KUKA KRL program: FINA11.src

&ACCESS RVP
&REL 143
DEF FINA11()
   DECL E6axis PX1 ;shengming px1 bianliang

   GLOBAL INTERRUPT DECL 3 WHEN $STOPMESS==TRUE DO IR_STOPM ( )
   INTERRUPT ON 3
   BAS (#INITMOV,0)
   BAS (#VEL_PTP,20)
   BAS (#ACC_PTP,20)
   $APO.CDIS = 100.0
   $VEL.CP = 0.5
   $ADVANCE=5
   $TOOL={X 0, Y 0, Z 319.5, A 0, B 0, C 0}
   $BASE={X 1708, Y 89, Z 1050, A 180, B 0, C 180}
   PTP {A1 -30.000, A2 -120.000, A3 120.000, A4 0.000, A5 0.000, A6 0.000, E1 0, E2 0, E3 0, E4 0, E5 0, E6 0}
   $async_EX_AX_DECOUPLE='b0001' ;dianji qu ouhe
   $AXIS_ACT.E1=0 ;bianmqi qingling
   WAIT SEC 1 ; yanshi 1s
   $async_EX_AX_DECOUPLE='b0000' ;dianji ouhe
   HALT
   $advance=5
   $VEL.CP=0.167
   $APO.CDIS = 0
   CONTINUE ;dongzuo lianguan
   ;IF SELT_MODE==1 THEN
   PTP {A1 5, A2 -84.46, A3 114.11, A4 59.82, A5 -48.27, A6 67.3, E1 0, E2 0, E3 0, E4 0, E5 0, E6 0} ;fenxian weizhi
   PTP {A1 5, A2 -84.46, A3 114.11, A4 59.82, A5 -48.27, A6 67.3, E1 0, E2 0, E3 0, E4 0, E5 0, E6 0} ;fenxian weizhi
   HALT ;zanting
   $APO.CDIS = 100 ;yuanhuaguodu
   PX1=$AXIS_ACT ;jiang dang qian jiaodu fuzhi gei px1
   NUM_TURN=1  ;zhuan jiao du ji shu bian liang
   CONTINUE
   $VEL.CP=0.167
   FOR NUM_TURN=1 TO 30  ;jiang NUM_TURN bianliang xunhuan 10ci
      PX1.E1=PX1.E1+120.0
      PTP PX1 C_DIS ;
   ENDFOR
   ;zan ting
   HALT
   ;PTP {A1 2.39, A2 -82.14, A3 104.12, A4 65.48, A5 -43.86, A6 58.47, E1 -84.06, E2 0, E3 0, E4 0, E5 0, E6 0}

   ;ELSE
   ;PTP {A1 7.433, A2 -36.447, A3 70.255, A4 38.782, A5 -95.202, A6 0.000, E1 -55.75, E2 0, E3 0, E4 0, E5 0, E6 0}
   ;SPTP {A1 7.433, A2 -36.447, A3 70.255, A4 38.782, A5 -95.202, A6 0.000, E1 -55.75, E2 0, E3 0, E4 0, E5 0, E6 0} C_DIS
   ;Start
   $VEL.CP=0.133
   SPTP {A1 7.880, A2 -36.991, A3 70.406, A4 40.976, A5 -94.486, A6 0.000, E1 -55.64, E2 0, E3 0, E4 0, E5 0, E6 0} C_DIS
   SPTP {A1 8.283, A2 -37.781, A3 70.980, A4 43.029, A5 -93.598, A6 0.000, E1 -55.77, E2 0, E3 0, E4 0, E5 0, E6 0} C_DIS
   SPTP {A1 8.645, A2 -38.809, A3 71.949, A4 44.960, A5 -92.527, A6 0.000, E1 -56.19, E2 0, E3 0, E4 0, E5 0, E6 0} C_DIS
   SPTP {A1 9.000, A2 -39.796, A3 72.797, A4 46.914, A5 -91.440, A6 0.000, E1 -56.68, E2 0, E3 0, E4 0, E5 0, E6 0} C_DIS
   SPTP {A1 9.348, A2 -40.751, A3 73.545, A4 48.891, A5 -90.338, A6 0.000, E1 -57.25, E2 0, E3 0, E4 0, E5 0, E6 0} C_DIS
   SPTP {A1 9.684, A2 -41.681, A3 74.210, A4 50.878, A5 -89.222, A6 0.000, E1 -57.87, E2 0, E3 0, E4 0, E5 0, E6 0} C_DIS
   SPTP {A1 10.009, A2 -42.594, A3 74.803, A4 52.874, A5 -88.090, A6 0.000, E1 -58.54, E2 0, E3 0, E4 0, E5 0, E6 0} C_DIS
   SPTP {A1 10.320, A2 -43.493, A3 75.334, A4 54.874, A5 -86.941, A6 0.000, E1 -59.25, E2 0, E3 0, E4 0, E5 0, E6 0} C_DIS
   SPTP {A1 10.615, A2 -44.382, A3 75.814, A4 56.876, A5 -85.776, A6 0.000, E1 -60, E2 0, E3 0, E4 0, E5 0, E6 0} C_DIS
   SPTP {A1 10.870, A2 -45.375, A3 76.460, A4 58.776, A5 -84.526, A6 0.000, E1 -60.98, E2 0, E3 0, E4 0, E5 0, E6 0} C_DIS
   SPTP {A1 11.099, A2 -46.403, A3 77.133, A4 60.647, A5 -83.228, A6 0.000, E1 -62.08, E2 0, E3 0, E4 0, E5 0, E6 0} C_DIS
   SPTP {A1 11.315, A2 -47.400, A3 77.716, A4 62.556, A5 -81.937, A6 0.000, E1 -63.25, E2 0, E3 0, E4 0, E5 0, E6 0} C_DIS
   SPTP {A1 11.512, A2 -48.390, A3 78.250, A4 64.480, A5 -80.631, A6 0.000, E1 -64.49, E2 0, E3 0, E4 0, E5 0, E6 0} C_DIS
   SPTP {A1 11.690, A2 -49.362, A3 78.719, A4 66.433, A5 -79.325, A6 0.000, E1 -65.79, E2 0, E3 0, E4 0, E5 0, E6 0} C_DIS
   SPTP {A1 11.848, A2 -50.324, A3 79.141, A4 68.407, A5 -78.011, A6 0.000, E1 -67.16, E2 0, E3 0, E4 0, E5 0, E6 0} C_DIS
   SPTP {A1 11.984, A2 -51.273, A3 79.509, A4 70.411, A5 -76.698, A6 0.000, E1 -68.6, E2 0, E3 0, E4 0, E5 0, E6 0} C_DIS
   SPTP {A1 12.098, A2 -52.202, A3 79.819, A4 72.452, A5 -75.397, A6 0.000, E1 -70.12, E2 0, E3 0, E4 0, E5 0, E6 0} C_DIS
   SPTP {A1 12.187, A2 -53.119, A3 80.083, A4 74.527, A5 -74.100, A6 0.000, E1 -71.71, E2 0, E3 0, E4 0, E5 0, E6 0} C_DIS
   SPTP {A1 12.253, A2 -54.007, A3 80.279, A4 76.654, A5 -72.833, A6 0.000, E1 -73.4, E2 0, E3 0, E4 0, E5 0, E6 0} C_DIS
   SPTP {A1 12.292, A2 -54.883, A3 80.432, A4 78.822, A5 -71.578, A6 0.000, E1 -75.17, E2 0, E3 0, E4 0, E5 0, E6 0} C_DIS
   SPTP {A1 12.307, A2 -55.719, A3 80.506, A4 81.058, A5 -70.379, A6 0.000, E1 -77.05, E2 0, E3 0, E4 0, E5 0, E6 0} C_DIS
   SPTP {A1 12.293, A2 -56.537, A3 80.534, A4 83.344, A5 -69.206, A6 0.000, E1 -79.02, E2 0, E3 0, E4 0, E5 0, E6 0} C_DIS
   SPTP {A1 12.254, A2 -57.299, A3 80.488, A4 85.654, A5 -68.116, A6 0.000, E1 -81, E2 0, E3 0, E4 0, E5 0, E6 0} C_DIS
   SPTP {A1 12.184, A2 -57.979, A3 80.434, A4 87.746, A5 -67.107, A6 0.000, E1 -82.51, E2 0, E3 0, E4 0, E5 0, E6 0} C_DIS
   HALT
   SPTP {A1 12.090, A2 -58.636, A3 80.350, A4 89.865, A5 -66.133, A6 0.000, E1 -84.06, E2 0, E3 0, E4 0, E5 0, E6 0} C_DIS
   SPTP {A1 11.972, A2 -59.275, A3 80.235, A4 92.031, A5 -65.193, A6 0.000, E1 -85.68, E2 0, E3 0, E4 0, E5 0, E6 0} C_DIS
   SPTP {A1 11.830, A2 -59.891, A3 80.084, A4 94.249, A5 -64.297, A6 0.000, E1 -87.37, E2 0, E3 0, E4 0, E5 0, E6 0} C_DIS
   SPTP {A1 11.665, A2 -60.478, A3 79.890, A4 96.525, A5 -63.457, A6 0.000, E1 -89.15, E2 0, E3 0, E4 0, E5 0, E6 0} C_DIS
   SPTP {A1 11.477, A2 -61.034, A3 79.651, A4 98.858, A5 -62.682, A6 0.000, E1 -91.01, E2 0, E3 0, E4 0, E5 0, E6 0} C_DIS
   SPTP {A1 11.269, A2 -61.552, A3 79.358, A4 101.252, A5 -61.990, A6 0.000, E1 -92.95, E2 0, E3 0, E4 0, E5 0, E6 0} C_DIS
   SPTP {A1 11.041, A2 -62.032, A3 79.039, A4 103.636, A5 -61.365, A6 0.000, E1 -94.82, E2 0, E3 0, E4 0, E5 0, E6 0} C_DIS
   SPTP {A1 10.795, A2 -62.519, A3 78.970, A4 105.496, A5 -60.574, A6 0.000, E1 -95.67, E2 0, E3 0, E4 0, E5 0, E6 0} C_DIS
   SPTP {A1 10.532, A2 -62.995, A3 78.892, A4 107.395, A5 -59.807, A6 0.000, E1 -96.57, E2 0, E3 0, E4 0, E5 0, E6 0} C_DIS
   SPTP {A1 10.254, A2 -63.455, A3 78.799, A4 109.336, A5 -59.075, A6 0.000, E1 -97.51, E2 0, E3 0, E4 0, E5 0, E6 0} C_DIS
   SPTP {A1 9.963, A2 -63.890, A3 78.682, A4 111.320, A5 -58.395, A6 0.000, E1 -98.5, E2 0, E3 0, E4 0, E5 0, E6 0} C_DIS
   SPTP {A1 9.661, A2 -64.298, A3 78.535, A4 113.347, A5 -57.779, A6 0.000, E1 -99.53, E2 0, E3 0, E4 0, E5 0, E6 0} C_DIS
   SPTP {A1 9.351, A2 -64.674, A3 78.354, A4 115.414, A5 -57.239, A6 0.000, E1 -100.59, E2 0, E3 0, E4 0, E5 0, E6 0} C_DIS
   SPTP {A1 9.036, A2 -65.116, A3 78.480, A4 117.001, A5 -56.418, A6 0.000, E1 -100.81, E2 0, E3 0, E4 0, E5 0, E6 0} C_DIS
   SPTP {A1 8.718, A2 -65.623, A3 78.879, A4 118.187, A5 -55.327, A6 0.000, E1 -100.36, E2 0, E3 0, E4 0, E5 0, E6 0} C_DIS
   SPTP {A1 8.399, A2 -66.115, A3 79.274, A4 119.383, A5 -54.253, A6 0.000, E1 -99.91, E2 0, E3 0, E4 0, E5 0, E6 0} C_DIS
   SPTP {A1 8.080, A2 -66.590, A3 79.662, A4 120.587, A5 -53.203, A6 0.000, E1 -99.46, E2 0, E3 0, E4 0, E5 0, E6 0} C_DIS
   SPTP {A1 7.762, A2 -67.048, A3 80.044, A4 121.798, A5 -52.179, A6 0.000, E1 -99.01, E2 0, E3 0, E4 0, E5 0, E6 0} C_DIS
   SPTP {A1 7.452, A2 -67.536, A3 80.590, A4 122.724, A5 -50.992, A6 0.000, E1 -98.13, E2 0, E3 0, E4 0, E5 0, E6 0} C_DIS
   SPTP {A1 7.154, A2 -68.181, A3 81.750, A4 122.572, A5 -49.106, A6 0.000, E1 -95.74, E2 0, E3 0, E4 0, E5 0, E6 0} C_DIS
   SPTP {A1 6.864, A2 -68.792, A3 82.894, A4 122.305, A5 -47.234, A6 0.000, E1 -93.25, E2 0, E3 0, E4 0, E5 0, E6 0} C_DIS
   SPTP {A1 6.585, A2 -69.369, A3 84.019, A4 121.908, A5 -45.386, A6 0.000, E1 -90.65, E2 0, E3 0, E4 0, E5 0, E6 0} C_DIS
   SPTP {A1 6.318, A2 -69.912, A3 85.124, A4 121.367, A5 -43.568, A6 0.000, E1 -87.91, E2 0, E3 0, E4 0, E5 0, E6 0} C_DIS
   SPTP {A1 6.068, A2 -70.459, A3 86.414, A4 120.139, A5 -41.551, A6 0.000, E1 -84.38, E2 0, E3 0, E4 0, E5 0, E6 0} C_DIS
   SPTP {A1 5.835, A2 -71.046, A3 88.208, A4 117.103, A5 -39.004, A6 0.000, E1 -78.78, E2 0, E3 0, E4 0, E5 0, E6 0} C_DIS
   SPTP {A1 5.615, A2 -71.534, A3 89.916, A4 113.493, A5 -36.647, A6 0.000, E1 -72.65, E2 0, E3 0, E4 0, E5 0, E6 0} C_DIS
   SPTP {A1 5.408, A2 -71.925, A3 91.535, A4 109.257, A5 -34.526, A6 0.000, E1 -65.93, E2 0, E3 0, E4 0, E5 0, E6 0} C_DIS
   SPTP {A1 5.213, A2 -72.216, A3 93.061, A4 104.367, A5 -32.693, A6 0.000, E1 -58.59, E2 0, E3 0, E4 0, E5 0, E6 0} C_DIS
   SPTP {A1 5.032, A2 -72.407, A3 94.490, A4 98.837, A5 -31.209, A6 0.000, E1 -50.64, E2 0, E3 0, E4 0, E5 0, E6 0} C_DIS
   SPTP {A1 4.862, A2 -72.471, A3 95.949, A4 91.902, A5 -30.163, A6 0.000, E1 -41.35, E2 0, E3 0, E4 0, E5 0, E6 0} C_DIS
   SPTP {A1 4.701, A2 -72.389, A3 97.348, A4 84.053, A5 -29.733, A6 0.000, E1 -31.19, E2 0, E3 0, E4 0, E5 0, E6 0} C_DIS
   SPTP {A1 4.547, A2 -72.174, A3 98.598, A4 76.137, A5 -29.944, A6 0.000, E1 -20.99, E2 0, E3 0, E4 0, E5 0, E6 0} C_DIS
   SPTP {A1 4.399, A2 -71.829, A3 99.695, A4 68.521, A5 -30.775, A6 0.000, E1 -11.11, E2 0, E3 0, E4 0, E5 0, E6 0} C_DIS
   SPTP {A1 4.261, A2 -71.353, A3 100.632, A4 61.519, A5 -32.180, A6 0.000, E1 -1.84, E2 0, E3 0, E4 0, E5 0, E6 0} C_DIS
   SPTP {A1 4.136, A2 -70.751, A3 101.404, A4 55.307, A5 -34.070, A6 0.000, E1 6.63, E2 0, E3 0, E4 0, E5 0, E6 0} C_DIS
   SPTP {A1 4.022, A2 -70.030, A3 102.012, A4 49.932, A5 -36.348, A6 0.000, E1 14.27, E2 0, E3 0, E4 0, E5 0, E6 0} C_DIS
   SPTP {A1 3.922, A2 -69.194, A3 102.450, A4 45.377, A5 -38.927, A6 0.000, E1 21.11, E2 0, E3 0, E4 0, E5 0, E6 0} C_DIS
   SPTP {A1 3.840, A2 -68.251, A3 102.716, A4 41.575, A5 -41.730, A6 0.000, E1 27.21, E2 0, E3 0, E4 0, E5 0, E6 0} C_DIS
   SPTP {A1 3.776, A2 -67.320, A3 102.827, A4 38.663, A5 -44.407, A6 0.000, E1 32.35, E2 0, E3 0, E4 0, E5 0, E6 0} C_DIS
   SPTP {A1 3.725, A2 -66.575, A3 102.861, A4 36.670, A5 -46.536, A6 0.000, E1 36.37, E2 0, E3 0, E4 0, E5 0, E6 0} C_DIS
   SPTP {A1 3.694, A2 -65.782, A3 102.799, A4 34.989, A5 -48.712, A6 0.000, E1 40.11, E2 0, E3 0, E4 0, E5 0, E6 0} C_DIS
   SPTP {A1 3.683, A2 -64.947, A3 102.644, A4 33.590, A5 -50.918, A6 0.000, E1 43.61, E2 0, E3 0, E4 0, E5 0, E6 0} C_DIS
   SPTP {A1 3.692, A2 -64.071, A3 102.395, A4 32.447, A5 -53.136, A6 0.000, E1 46.88, E2 0, E3 0, E4 0, E5 0, E6 0} C_DIS
   SPTP {A1 3.720, A2 -63.161, A3 102.055, A4 31.529, A5 -55.351, A6 0.000, E1 49.96, E2 0, E3 0, E4 0, E5 0, E6 0} C_DIS
   SPTP {A1 3.765, A2 -62.219, A3 101.624, A4 30.813, A5 -57.551, A6 0.000, E1 52.88, E2 0, E3 0, E4 0, E5 0, E6 0} C_DIS
   SPTP {A1 3.868, A2 -61.648, A3 101.314, A4 30.672, A5 -58.896, A6 0.000, E1 55.21, E2 0, E3 0, E4 0, E5 0, E6 0} C_DIS
   SPTP {A1 3.996, A2 -61.138, A3 100.997, A4 30.721, A5 -60.077, A6 0.000, E1 57.38, E2 0, E3 0, E4 0, E5 0, E6 0} C_DIS
   SPTP {A1 4.141, A2 -60.619, A3 100.641, A4 30.875, A5 -61.247, A6 0.000, E1 59.47, E2 0, E3 0, E4 0, E5 0, E6 0} C_DIS
   SPTP {A1 4.300, A2 -60.092, A3 100.246, A4 31.122, A5 -62.400, A6 0.000, E1 61.49, E2 0, E3 0, E4 0, E5 0, E6 0} C_DIS
   SPTP {A1 4.471, A2 -59.559, A3 99.814, A4 31.448, A5 -63.534, A6 0.000, E1 63.46, E2 0, E3 0, E4 0, E5 0, E6 0} C_DIS
   SPTP {A1 4.653, A2 -59.019, A3 99.345, A4 31.854, A5 -64.648, A6 0.000, E1 65.37, E2 0, E3 0, E4 0, E5 0, E6 0} C_DIS
   SPTP {A1 4.843, A2 -58.475, A3 98.842, A4 32.326, A5 -65.738, A6 0.000, E1 67.23, E2 0, E3 0, E4 0, E5 0, E6 0} C_DIS
   SPTP {A1 5.048, A2 -57.962, A3 98.326, A4 32.894, A5 -66.735, A6 0.000, E1 69.02, E2 0, E3 0, E4 0, E5 0, E6 0} C_DIS
   SPTP {A1 5.321, A2 -57.796, A3 98.000, A4 33.874, A5 -67.052, A6 0.000, E1 70.48, E2 0, E3 0, E4 0, E5 0, E6 0} C_DIS
   SPTP {A1 5.599, A2 -57.626, A3 97.650, A4 34.901, A5 -67.358, A6 0.000, E1 71.89, E2 0, E3 0, E4 0, E5 0, E6 0} C_DIS
   SPTP {A1 5.882, A2 -57.453, A3 97.275, A4 35.972, A5 -67.654, A6 0.000, E1 73.26, E2 0, E3 0, E4 0, E5 0, E6 0} C_DIS
   SPTP {A1 6.166, A2 -57.278, A3 96.877, A4 37.078, A5 -67.938, A6 0.000, E1 74.59, E2 0, E3 0, E4 0, E5 0, E6 0} C_DIS
   SPTP {A1 6.452, A2 -57.099, A3 96.455, A4 38.215, A5 -68.213, A6 0.000, E1 75.9, E2 0, E3 0, E4 0, E5 0, E6 0} C_DIS
   SPTP {A1 6.737, A2 -56.918, A3 96.010, A4 39.378, A5 -68.477, A6 0.000, E1 77.18, E2 0, E3 0, E4 0, E5 0, E6 0} C_DIS
   SPTP {A1 7.020, A2 -56.735, A3 95.545, A4 40.563, A5 -68.731, A6 0.000, E1 78.43, E2 0, E3 0, E4 0, E5 0, E6 0} C_DIS
   SPTP {A1 7.301, A2 -56.550, A3 95.058, A4 41.765, A5 -68.973, A6 0.000, E1 79.67, E2 0, E3 0, E4 0, E5 0, E6 0} C_DIS
   SPTP {A1 7.577, A2 -56.363, A3 94.553, A4 42.980, A5 -69.205, A6 0.000, E1 80.88, E2 0, E3 0, E4 0, E5 0, E6 0} C_DIS
   SPTP {A1 7.849, A2 -56.176, A3 94.029, A4 44.204, A5 -69.426, A6 0.000, E1 82.08, E2 0, E3 0, E4 0, E5 0, E6 0} C_DIS
   SPTP {A1 8.115, A2 -55.987, A3 93.489, A4 45.437, A5 -69.637, A6 0.000, E1 83.27, E2 0, E3 0, E4 0, E5 0, E6 0} C_DIS
   SPTP {A1 8.380, A2 -55.851, A3 92.971, A4 46.723, A5 -69.748, A6 0.000, E1 84.36, E2 0, E3 0, E4 0, E5 0, E6 0} C_DIS
   SPTP {A1 8.645, A2 -55.786, A3 92.489, A4 48.086, A5 -69.733, A6 0.000, E1 85.33, E2 0, E3 0, E4 0, E5 0, E6 0} C_DIS
   SPTP {A1 8.902, A2 -55.719, A3 91.992, A4 49.451, A5 -69.712, A6 0.000, E1 86.28, E2 0, E3 0, E4 0, E5 0, E6 0} C_DIS
   SPTP {A1 9.152, A2 -55.650, A3 91.480, A4 50.817, A5 -69.688, A6 0.000, E1 87.22, E2 0, E3 0, E4 0, E5 0, E6 0} C_DIS
   SPTP {A1 9.393, A2 -55.581, A3 90.956, A4 52.180, A5 -69.658, A6 0.000, E1 88.15, E2 0, E3 0, E4 0, E5 0, E6 0} C_DIS
   SPTP {A1 9.624, A2 -55.511, A3 90.422, A4 53.538, A5 -69.624, A6 0.000, E1 89.08, E2 0, E3 0, E4 0, E5 0, E6 0} C_DIS
   SPTP {A1 9.845, A2 -55.443, A3 89.880, A4 54.890, A5 -69.583, A6 0.000, E1 90, E2 0, E3 0, E4 0, E5 0, E6 0} C_DIS
   SPTP {A1 10.057, A2 -55.377, A3 89.331, A4 56.233, A5 -69.536, A6 0.000, E1 90.92, E2 0, E3 0, E4 0, E5 0, E6 0} C_DIS
   SPTP {A1 10.258, A2 -55.314, A3 88.779, A4 57.563, A5 -69.480, A6 0.000, E1 91.84, E2 0, E3 0, E4 0, E5 0, E6 0} C_DIS
   SPTP {A1 10.448, A2 -55.255, A3 88.225, A4 58.882, A5 -69.417, A6 0.000, E1 92.76, E2 0, E3 0, E4 0, E5 0, E6 0} C_DIS
   SPTP {A1 10.623, A2 -55.202, A3 87.683, A4 60.164, A5 -69.349, A6 0.000, E1 93.68, E2 0, E3 0, E4 0, E5 0, E6 0} C_DIS
   SPTP {A1 10.779, A2 -55.156, A3 87.166, A4 61.385, A5 -69.290, A6 0.000, E1 94.58, E2 0, E3 0, E4 0, E5 0, E6 0} C_DIS
   SPTP {A1 10.910, A2 -55.118, A3 86.689, A4 62.513, A5 -69.244, A6 0.000, E1 95.46, E2 0, E3 0, E4 0, E5 0, E6 0} C_DIS
   SPTP {A1 11.018, A2 -55.088, A3 86.256, A4 63.546, A5 -69.214, A6 0.000, E1 96.32, E2 0, E3 0, E4 0, E5 0, E6 0} C_DIS
   SPTP {A1 11.118, A2 -55.067, A3 85.835, A4 64.562, A5 -69.171, A6 0.000, E1 97.19, E2 0, E3 0, E4 0, E5 0, E6 0} C_DIS
   SPTP {A1 11.209, A2 -55.057, A3 85.426, A4 65.558, A5 -69.111, A6 0.000, E1 98.08, E2 0, E3 0, E4 0, E5 0, E6 0} C_DIS
   SPTP {A1 11.292, A2 -55.060, A3 85.035, A4 66.532, A5 -69.032, A6 0.000, E1 98.98, E2 0, E3 0, E4 0, E5 0, E6 0} C_DIS
   SPTP {A1 11.366, A2 -55.075, A3 84.661, A4 67.487, A5 -68.936, A6 0.000, E1 99.9, E2 0, E3 0, E4 0, E5 0, E6 0} C_DIS
   SPTP {A1 11.432, A2 -55.102, A3 84.304, A4 68.421, A5 -68.820, A6 0.000, E1 100.83, E2 0, E3 0, E4 0, E5 0, E6 0} C_DIS
   SPTP {A1 11.490, A2 -55.143, A3 83.969, A4 69.335, A5 -68.684, A6 0.000, E1 101.78, E2 0, E3 0, E4 0, E5 0, E6 0} C_DIS
   SPTP {A1 11.539, A2 -55.199, A3 83.655, A4 70.227, A5 -68.526, A6 0.000, E1 102.74, E2 0, E3 0, E4 0, E5 0, E6 0} C_DIS
   SPTP {A1 11.581, A2 -55.269, A3 83.364, A4 71.100, A5 -68.347, A6 0.000, E1 103.72, E2 0, E3 0, E4 0, E5 0, E6 0} C_DIS
   SPTP {A1 11.614, A2 -55.358, A3 83.100, A4 71.948, A5 -68.140, A6 0.000, E1 104.71, E2 0, E3 0, E4 0, E5 0, E6 0} C_DIS
   SPTP {A1 11.638, A2 -55.462, A3 82.861, A4 72.775, A5 -67.908, A6 0.000, E1 105.72, E2 0, E3 0, E4 0, E5 0, E6 0} C_DIS
   SPTP {A1 11.655, A2 -55.583, A3 82.649, A4 73.581, A5 -67.651, A6 0.000, E1 106.75, E2 0, E3 0, E4 0, E5 0, E6 0} C_DIS
   SPTP {A1 11.664, A2 -55.722, A3 82.465, A4 74.365, A5 -67.366, A6 0.000, E1 107.8, E2 0, E3 0, E4 0, E5 0, E6 0} C_DIS
   SPTP {A1 11.664, A2 -55.877, A3 82.310, A4 75.127, A5 -67.054, A6 0.000, E1 108.86, E2 0, E3 0, E4 0, E5 0, E6 0} C_DIS
   SPTP {A1 11.657, A2 -56.050, A3 82.184, A4 75.868, A5 -66.713, A6 0.000, E1 109.94, E2 0, E3 0, E4 0, E5 0, E6 0} C_DIS
   SPTP {A1 11.642, A2 -56.241, A3 82.087, A4 76.588, A5 -66.342, A6 0.000, E1 111.03, E2 0, E3 0, E4 0, E5 0, E6 0} C_DIS
   SPTP {A1 11.614, A2 -56.480, A3 82.054, A4 77.308, A5 -65.925, A6 0.000, E1 111.95, E2 0, E3 0, E4 0, E5 0, E6 0} C_DIS
   SPTP {A1 11.575, A2 -56.756, A3 82.072, A4 78.027, A5 -65.467, A6 0.000, E1 112.75, E2 0, E3 0, E4 0, E5 0, E6 0} C_DIS
   SPTP {A1 11.529, A2 -57.044, A3 82.112, A4 78.732, A5 -64.986, A6 0.000, E1 113.55, E2 0, E3 0, E4 0, E5 0, E6 0} C_DIS
   SPTP {A1 11.475, A2 -57.347, A3 82.174, A4 79.421, A5 -64.478, A6 0.000, E1 114.36, E2 0, E3 0, E4 0, E5 0, E6 0} C_DIS
   SPTP {A1 11.413, A2 -57.663, A3 82.259, A4 80.095, A5 -63.943, A6 0.000, E1 115.18, E2 0, E3 0, E4 0, E5 0, E6 0} C_DIS
   SPTP {A1 11.344, A2 -57.991, A3 82.364, A4 80.756, A5 -63.383, A6 0.000, E1 116, E2 0, E3 0, E4 0, E5 0, E6 0} C_DIS
   SPTP {A1 11.267, A2 -58.332, A3 82.492, A4 81.402, A5 -62.796, A6 0.000, E1 116.83, E2 0, E3 0, E4 0, E5 0, E6 0} C_DIS
   SPTP {A1 11.182, A2 -58.686, A3 82.641, A4 82.033, A5 -62.180, A6 0.000, E1 117.67, E2 0, E3 0, E4 0, E5 0, E6 0} C_DIS
   SPTP {A1 11.089, A2 -59.052, A3 82.812, A4 82.650, A5 -61.536, A6 0.000, E1 118.51, E2 0, E3 0, E4 0, E5 0, E6 0} C_DIS
   SPTP {A1 10.987, A2 -59.430, A3 83.003, A4 83.253, A5 -60.864, A6 0.000, E1 119.35, E2 0, E3 0, E4 0, E5 0, E6 0} C_DIS
   SPTP {A1 10.877, A2 -59.819, A3 83.215, A4 83.842, A5 -60.164, A6 0.000, E1 120.2, E2 0, E3 0, E4 0, E5 0, E6 0} C_DIS
   SPTP {A1 10.759, A2 -60.218, A3 83.445, A4 84.418, A5 -59.436, A6 0.000, E1 121.05, E2 0, E3 0, E4 0, E5 0, E6 0} C_DIS
   SPTP {A1 10.638, A2 -60.676, A3 83.610, A4 85.382, A5 -58.579, A6 0.000, E1 121.44, E2 0, E3 0, E4 0, E5 0, E6 0} C_DIS
   SPTP {A1 10.508, A2 -61.154, A3 83.752, A4 86.490, A5 -57.675, A6 0.000, E1 121.67, E2 0, E3 0, E4 0, E5 0, E6 0} C_DIS
   SPTP {A1 10.366, A2 -61.633, A3 83.899, A4 87.611, A5 -56.757, A6 0.000, E1 121.87, E2 0, E3 0, E4 0, E5 0, E6 0} C_DIS
   SPTP {A1 10.212, A2 -62.114, A3 84.052, A4 88.745, A5 -55.824, A6 0.000, E1 122.04, E2 0, E3 0, E4 0, E5 0, E6 0} C_DIS
   SPTP {A1 10.047, A2 -62.596, A3 84.209, A4 89.896, A5 -54.879, A6 0.000, E1 122.18, E2 0, E3 0, E4 0, E5 0, E6 0} C_DIS
   SPTP {A1 9.870, A2 -63.077, A3 84.370, A4 91.065, A5 -53.921, A6 0.000, E1 122.29, E2 0, E3 0, E4 0, E5 0, E6 0} C_DIS
   SPTP {A1 9.681, A2 -63.559, A3 84.534, A4 92.254, A5 -52.951, A6 0.000, E1 122.37, E2 0, E3 0, E4 0, E5 0, E6 0} C_DIS
   SPTP {A1 9.479, A2 -64.040, A3 84.702, A4 93.467, A5 -51.971, A6 0.000, E1 122.41, E2 0, E3 0, E4 0, E5 0, E6 0} C_DIS
   SPTP {A1 9.265, A2 -64.519, A3 84.872, A4 94.705, A5 -50.979, A6 0.000, E1 122.41, E2 0, E3 0, E4 0, E5 0, E6 0} C_DIS
   SPTP {A1 9.039, A2 -64.997, A3 85.045, A4 95.972, A5 -49.979, A6 0.000, E1 122.37, E2 0, E3 0, E4 0, E5 0, E6 0} C_DIS
   SPTP {A1 8.801, A2 -65.471, A3 85.217, A4 97.272, A5 -48.973, A6 0.000, E1 122.29, E2 0, E3 0, E4 0, E5 0, E6 0} C_DIS
   SPTP {A1 8.551, A2 -65.941, A3 85.390, A4 98.607, A5 -47.961, A6 0.000, E1 122.16, E2 0, E3 0, E4 0, E5 0, E6 0} C_DIS
   SPTP {A1 8.289, A2 -66.407, A3 85.564, A4 99.981, A5 -46.943, A6 0.000, E1 121.98, E2 0, E3 0, E4 0, E5 0, E6 0} C_DIS
   SPTP {A1 8.015, A2 -66.868, A3 85.736, A4 101.397, A5 -45.924, A6 0.000, E1 121.75, E2 0, E3 0, E4 0, E5 0, E6 0} C_DIS
   SPTP {A1 7.730, A2 -67.322, A3 85.903, A4 102.871, A5 -44.907, A6 0.000, E1 121.46, E2 0, E3 0, E4 0, E5 0, E6 0} C_DIS
   SPTP {A1 7.416, A2 -67.782, A3 85.963, A4 104.870, A5 -43.810, A6 0.000, E1 120.85, E2 0, E3 0, E4 0, E5 0, E6 0} C_DIS
   SPTP {A1 7.087, A2 -68.230, A3 86.018, A4 106.947, A5 -42.736, A6 0.000, E1 120.16, E2 0, E3 0, E4 0, E5 0, E6 0} C_DIS
   SPTP {A1 6.744, A2 -68.667, A3 86.069, A4 109.106, A5 -41.681, A6 0.000, E1 119.38, E2 0, E3 0, E4 0, E5 0, E6 0} C_DIS
   SPTP {A1 6.387, A2 -69.092, A3 86.117, A4 111.353, A5 -40.653, A6 0.000, E1 118.51, E2 0, E3 0, E4 0, E5 0, E6 0} C_DIS
   SPTP {A1 6.016, A2 -69.504, A3 86.160, A4 113.693, A5 -39.654, A6 0.000, E1 117.53, E2 0, E3 0, E4 0, E5 0, E6 0} C_DIS
   SPTP {A1 5.633, A2 -69.902, A3 86.197, A4 116.128, A5 -38.693, A6 0.000, E1 116.46, E2 0, E3 0, E4 0, E5 0, E6 0} C_DIS
   SPTP {A1 5.238, A2 -70.285, A3 86.228, A4 118.661, A5 -37.776, A6 0.000, E1 115.28, E2 0, E3 0, E4 0, E5 0, E6 0} C_DIS
   SPTP {A1 4.833, A2 -70.651, A3 86.253, A4 121.291, A5 -36.910, A6 0.000, E1 114.01, E2 0, E3 0, E4 0, E5 0, E6 0} C_DIS
   SPTP {A1 4.420, A2 -71.001, A3 86.271, A4 124.016, A5 -36.101, A6 0.000, E1 112.65, E2 0, E3 0, E4 0, E5 0, E6 0} C_DIS
   SPTP {A1 3.999, A2 -71.335, A3 86.281, A4 126.833, A5 -35.354, A6 0.000, E1 111.19, E2 0, E3 0, E4 0, E5 0, E6 0} C_DIS
   SPTP {A1 3.573, A2 -71.651, A3 86.285, A4 129.733, A5 -34.676, A6 0.000, E1 109.67, E2 0, E3 0, E4 0, E5 0, E6 0} C_DIS
   SPTP {A1 3.142, A2 -71.950, A3 86.283, A4 132.707, A5 -34.069, A6 0.000, E1 108.07, E2 0, E3 0, E4 0, E5 0, E6 0} C_DIS
   SPTP {A1 2.710, A2 -72.231, A3 86.274, A4 135.737, A5 -33.543, A6 0.000, E1 106.44, E2 0, E3 0, E4 0, E5 0, E6 0} C_DIS
   SPTP {A1 2.276, A2 -72.545, A3 86.443, A4 138.426, A5 -32.805, A6 0.000, E1 105.24, E2 0, E3 0, E4 0, E5 0, E6 0} C_DIS
   SPTP {A1 1.842, A2 -72.917, A3 86.884, A4 140.630, A5 -31.677, A6 0.000, E1 104.67, E2 0, E3 0, E4 0, E5 0, E6 0} C_DIS
   SPTP {A1 1.410, A2 -73.278, A3 87.332, A4 142.908, A5 -30.574, A6 0.000, E1 104.02, E2 0, E3 0, E4 0, E5 0, E6 0} C_DIS
   SPTP {A1 0.985, A2 -73.627, A3 87.785, A4 145.255, A5 -29.501, A6 0.000, E1 103.32, E2 0, E3 0, E4 0, E5 0, E6 0} C_DIS
   SPTP {A1 0.571, A2 -73.964, A3 88.245, A4 147.658, A5 -28.464, A6 0.000, E1 102.57, E2 0, E3 0, E4 0, E5 0, E6 0} C_DIS
   SPTP {A1 0.170, A2 -74.289, A3 88.711, A4 150.100, A5 -27.464, A6 0.000, E1 101.81, E2 0, E3 0, E4 0, E5 0, E6 0} C_DIS
   SPTP {A1 -0.212, A2 -74.603, A3 89.185, A4 152.558, A5 -26.503, A6 0.000, E1 101.05, E2 0, E3 0, E4 0, E5 0, E6 0} C_DIS
   SPTP {A1 -0.568, A2 -74.941, A3 89.813, A4 154.670, A5 -25.309, A6 0.000, E1 100.67, E2 0, E3 0, E4 0, E5 0, E6 0} C_DIS
   SPTP {A1 -0.886, A2 -75.387, A3 91.014, A4 155.445, A5 -23.052, A6 0.000, E1 101.64, E2 0, E3 0, E4 0, E5 0, E6 0} C_DIS
   SPTP {A1 -1.174, A2 -75.798, A3 92.198, A4 156.083, A5 -20.795, A6 0.000, E1 102.75, E2 0, E3 0, E4 0, E5 0, E6 0} C_DIS
   SPTP {A1 -1.424, A2 -76.174, A3 93.363, A4 156.463, A5 -18.550, A6 0.000, E1 104.14, E2 0, E3 0, E4 0, E5 0, E6 0} C_DIS
   SPTP {A1 -1.631, A2 -76.514, A3 94.509, A4 156.440, A5 -16.319, A6 0.000, E1 105.97, E2 0, E3 0, E4 0, E5 0, E6 0} C_DIS
   SPTP {A1 -1.784, A2 -76.833, A3 95.807, A4 154.943, A5 -13.728, A6 0.000, E1 109.29, E2 0, E3 0, E4 0, E5 0, E6 0} C_DIS
   SPTP {A1 -1.888, A2 -77.114, A3 97.660, A4 147.397, A5 -9.850, A6 0.000, E1 118.61, E2 0, E3 0, E4 0, E5 0, E6 0} C_DIS
   SPTP {A1 -1.939, A2 -77.267, A3 99.394, A4 129.667, A5 -6.466, A6 0.000, E1 138.11, E2 0, E3 0, E4 0, E5 0, E6 0} C_DIS
   SPTP {A1 -1.944, A2 -77.288, A3 101.004, A4 89.170, A5 -4.811, A6 0.000, E1 180.39, E2 0, E3 0, E4 0, E5 0, E6 0} C_DIS
   SPTP {A1 -1.886, A2 -77.175, A3 102.480, A4 48.596, A5 -6.473, A6 0.000, E1 222.77, E2 0, E3 0, E4 0, E5 0, E6 0} C_DIS
   SPTP {A1 -1.795, A2 -76.704, A3 104.251, A4 26.124, A5 -11.488, A6 0.000, E1 247.06, E2 0, E3 0, E4 0, E5 0, E6 0} C_DIS
   SPTP {A1 -1.664, A2 -75.882, A3 105.817, A4 17.958, A5 -17.686, A6 0.000, E1 257.05, E2 0, E3 0, E4 0, E5 0, E6 0} C_DIS
   SPTP {A1 -1.498, A2 -74.762, A3 107.020, A4 14.521, A5 -24.043, A6 0.000, E1 262.3, E2 0, E3 0, E4 0, E5 0, E6 0} C_DIS
   SPTP {A1 -1.315, A2 -73.120, A3 107.908, A4 12.419, A5 -31.256, A6 0.000, E1 266.34, E2 0, E3 0, E4 0, E5 0, E6 0} C_DIS
   SPTP {A1 -1.118, A2 -70.714, A3 108.276, A4 10.996, A5 -39.646, A6 0.000, E1 269.89, E2 0, E3 0, E4 0, E5 0, E6 0} C_DIS
   SPTP {A1 -0.922, A2 -67.914, A3 107.935, A4 10.302, A5 -47.764, A6 0.000, E1 272.72, E2 0, E3 0, E4 0, E5 0, E6 0} C_DIS
   SPTP {A1 -0.737, A2 -64.799, A3 106.887, A4 9.993, A5 -55.510, A6 0.000, E1 275.19, E2 0, E3 0, E4 0, E5 0, E6 0} C_DIS
   SPTP {A1 -0.488, A2 -61.717, A3 105.298, A4 10.147, A5 -62.262, A6 0.000, E1 277.55, E2 0, E3 0, E4 0, E5 0, E6 0} C_DIS
   SPTP {A1 -0.080, A2 -59.032, A3 103.499, A4 10.922, A5 -67.576, A6 0.000, E1 279.97, E2 0, E3 0, E4 0, E5 0, E6 0} C_DIS
   SPTP {A1 0.343, A2 -56.296, A3 101.299, A4 11.852, A5 -72.520, A6 0.000, E1 282.34, E2 0, E3 0, E4 0, E5 0, E6 0} C_DIS
   SPTP {A1 0.781, A2 -53.535, A3 98.716, A4 12.936, A5 -77.079, A6 0.000, E1 284.67, E2 0, E3 0, E4 0, E5 0, E6 0} C_DIS
   SPTP {A1 1.227, A2 -50.771, A3 95.770, A4 14.148, A5 -81.248, A6 0.000, E1 286.97, E2 0, E3 0, E4 0, E5 0, E6 0} C_DIS
   SPTP {A1 1.678, A2 -48.016, A3 92.477, A4 15.486, A5 -85.028, A6 0.000, E1 289.24, E2 0, E3 0, E4 0, E5 0, E6 0} C_DIS
   SPTP {A1 2.135, A2 -45.273, A3 88.843, A4 16.954, A5 -88.425, A6 0.000, E1 291.48, E2 0, E3 0, E4 0, E5 0, E6 0} C_DIS
   SPTP {A1 2.597, A2 -42.534, A3 84.865, A4 18.553, A5 -91.452, A6 0.000, E1 293.66, E2 0, E3 0, E4 0, E5 0, E6 0} C_DIS
   SPTP {A1 3.060, A2 -39.786, A3 80.534, A4 20.271, A5 -94.115, A6 0.000, E1 295.77, E2 0, E3 0, E4 0, E5 0, E6 0} C_DIS
   SPTP {A1 3.519, A2 -37.006, A3 75.823, A4 22.095, A5 -96.423, A6 0.000, E1 297.77, E2 0, E3 0, E4 0, E5 0, E6 0} C_DIS
   SPTP {A1 4.002, A2 -34.849, A3 71.834, A4 24.063, A5 -97.910, A6 0.000, E1 299.52, E2 0, E3 0, E4 0, E5 0, E6 0} C_DIS
   SPTP {A1 4.569, A2 -34.745, A3 71.119, A4 26.251, A5 -97.820, A6 0.000, E1 300.8, E2 0, E3 0, E4 0, E5 0, E6 0} C_DIS
   SPTP {A1 5.129, A2 -34.620, A3 70.315, A4 28.506, A5 -97.697, A6 0.000, E1 301.92, E2 0, E3 0, E4 0, E5 0, E6 0} C_DIS
   SPTP {A1 5.678, A2 -34.471, A3 69.415, A4 30.810, A5 -97.547, A6 0.000, E1 302.89, E2 0, E3 0, E4 0, E5 0, E6 0} C_DIS
   SPTP {A1 6.182, A2 -34.824, A3 69.368, A4 33.002, A5 -97.068, A6 0.000, E1 303.53, E2 0, E3 0, E4 0, E5 0, E6 0} C_DIS
   SPTP {A1 6.658, A2 -35.467, A3 69.798, A4 35.140, A5 -96.378, A6 0.000, E1 303.89, E2 0, E3 0, E4 0, E5 0, E6 0} C_DIS
   SPTP {A1 7.049, A2 -35.970, A3 70.064, A4 36.954, A5 -95.793, A6 0.000, E1 304.1, E2 0, E3 0, E4 0, E5 0, E6 0} C_DIS
   SPTP {A1 7.433, A2 -36.447, A3 70.255, A4 38.782, A5 -95.202, A6 0.000, E1 304.25, E2 0, E3 0, E4 0, E5 0, E6 0} C_DIS
   SPTP {A1 7.434, A2 -36.432, A3 70.237, A4 38.796, A5 -95.213, A6 0.000, E1 304.23, E2 0, E3 0, E4 0, E5 0, E6 0} C_DIS
   SPTP {A1 7.881, A2 -36.973, A3 70.384, A4 40.990, A5 -94.500, A6 0.000, E1 304.34, E2 0, E3 0, E4 0, E5 0, E6 0} C_DIS
   SPTP {A1 8.284, A2 -37.760, A3 70.952, A4 43.046, A5 -93.616, A6 0.000, E1 304.2, E2 0, E3 0, E4 0, E5 0, E6 0} C_DIS
   SPTP {A1 8.647, A2 -38.785, A3 71.916, A4 44.979, A5 -92.548, A6 0.000, E1 303.78, E2 0, E3 0, E4 0, E5 0, E6 0} C_DIS
   SPTP {A1 9.002, A2 -39.770, A3 72.763, A4 46.935, A5 -91.463, A6 0.000, E1 303.29, E2 0, E3 0, E4 0, E5 0, E6 0} C_DIS
   SPTP {A1 9.349, A2 -40.724, A3 73.509, A4 48.913, A5 -90.363, A6 0.000, E1 302.72, E2 0, E3 0, E4 0, E5 0, E6 0} C_DIS
   SPTP {A1 9.686, A2 -41.653, A3 74.171, A4 50.901, A5 -89.249, A6 0.000, E1 302.1, E2 0, E3 0, E4 0, E5 0, E6 0} C_DIS
   SPTP {A1 10.011, A2 -42.565, A3 74.763, A4 52.897, A5 -88.119, A6 0.000, E1 301.43, E2 0, E3 0, E4 0, E5 0, E6 0} C_DIS
   SPTP {A1 10.322, A2 -43.462, A3 75.294, A4 54.897, A5 -86.973, A6 0.000, E1 300.72, E2 0, E3 0, E4 0, E5 0, E6 0} C_DIS
   SPTP {A1 10.617, A2 -44.350, A3 75.772, A4 56.900, A5 -85.810, A6 0.000, E1 299.96, E2 0, E3 0, E4 0, E5 0, E6 0} C_DIS
   SPTP {A1 10.872, A2 -45.342, A3 76.417, A4 58.801, A5 -84.562, A6 0.000, E1 298.99, E2 0, E3 0, E4 0, E5 0, E6 0} C_DIS
   SPTP {A1 11.102, A2 -46.370, A3 77.089, A4 60.672, A5 -83.266, A6 0.000, E1 297.9, E2 0, E3 0, E4 0, E5 0, E6 0} C_DIS
   SPTP {A1 11.318, A2 -47.367, A3 77.673, A4 62.582, A5 -81.978, A6 0.000, E1 296.72, E2 0, E3 0, E4 0, E5 0, E6 0} C_DIS
   SPTP {A1 11.515, A2 -48.357, A3 78.206, A4 64.505, A5 -80.673, A6 0.000, E1 295.49, E2 0, E3 0, E4 0, E5 0, E6 0} C_DIS
   SPTP {A1 11.694, A2 -49.328, A3 78.676, A4 66.458, A5 -79.369, A6 0.000, E1 294.18, E2 0, E3 0, E4 0, E5 0, E6 0} C_DIS
   SPTP {A1 11.852, A2 -50.290, A3 79.098, A4 68.431, A5 -78.056, A6 0.000, E1 292.82, E2 0, E3 0, E4 0, E5 0, E6 0} C_DIS
   SPTP {A1 11.989, A2 -51.238, A3 79.467, A4 70.435, A5 -76.745, A6 0.000, E1 291.38, E2 0, E3 0, E4 0, E5 0, E6 0} C_DIS
   SPTP {A1 12.103, A2 -52.168, A3 79.777, A4 72.475, A5 -75.444, A6 0.000, E1 289.86, E2 0, E3 0, E4 0, E5 0, E6 0} C_DIS
   SPTP {A1 12.192, A2 -53.085, A3 80.042, A4 74.549, A5 -74.149, A6 0.000, E1 288.27, E2 0, E3 0, E4 0, E5 0, E6 0} C_DIS
   SPTP {A1 12.258, A2 -53.973, A3 80.239, A4 76.675, A5 -72.883, A6 0.000, E1 286.59, E2 0, E3 0, E4 0, E5 0, E6 0} C_DIS
   SPTP {A1 12.297, A2 -54.849, A3 80.393, A4 78.842, A5 -71.630, A6 0.000, E1 284.82, E2 0, E3 0, E4 0, E5 0, E6 0} C_DIS
   SPTP {A1 12.313, A2 -55.685, A3 80.468, A4 81.076, A5 -70.430, A6 0.000, E1 282.94, E2 0, E3 0, E4 0, E5 0, E6 0} C_DIS
   SPTP {A1 12.300, A2 -56.504, A3 80.498, A4 83.360, A5 -69.258, A6 0.000, E1 280.98, E2 0, E3 0, E4 0, E5 0, E6 0} C_DIS
   SPTP {A1 12.261, A2 -57.267, A3 80.454, A4 85.668, A5 -68.168, A6 0.000, E1 279, E2 0, E3 0, E4 0, E5 0, E6 0} C_DIS
   SPTP {A1 12.191, A2 -57.948, A3 80.401, A4 87.758, A5 -67.159, A6 0.000, E1 277.49, E2 0, E3 0, E4 0, E5 0, E6 0} C_DIS
   SPTP {A1 12.097, A2 -58.606, A3 80.319, A4 89.874, A5 -66.184, A6 0.000, E1 275.95, E2 0, E3 0, E4 0, E5 0, E6 0} C_DIS
   SPTP {A1 11.979, A2 -59.246, A3 80.205, A4 92.038, A5 -65.243, A6 0.000, E1 274.33, E2 0, E3 0, E4 0, E5 0, E6 0} C_DIS
   SPTP {A1 11.838, A2 -59.862, A3 80.056, A4 94.253, A5 -64.346, A6 0.000, E1 272.64, E2 0, E3 0, E4 0, E5 0, E6 0} C_DIS
   SPTP {A1 11.673, A2 -60.450, A3 79.864, A4 96.526, A5 -63.506, A6 0.000, E1 270.86, E2 0, E3 0, E4 0, E5 0, E6 0} C_DIS
   SPTP {A1 11.485, A2 -61.008, A3 79.628, A4 98.855, A5 -62.729, A6 0.000, E1 269.01, E2 0, E3 0, E4 0, E5 0, E6 0} C_DIS
   SPTP {A1 11.276, A2 -61.528, A3 79.337, A4 101.246, A5 -62.034, A6 0.000, E1 267.07, E2 0, E3 0, E4 0, E5 0, E6 0} C_DIS
   SPTP {A1 11.048, A2 -62.009, A3 79.019, A4 103.631, A5 -61.408, A6 0.000, E1 265.19, E2 0, E3 0, E4 0, E5 0, E6 0} C_DIS
   SPTP {A1 10.803, A2 -62.498, A3 78.952, A4 105.488, A5 -60.615, A6 0.000, E1 264.35, E2 0, E3 0, E4 0, E5 0, E6 0} C_DIS
   SPTP {A1 10.540, A2 -62.975, A3 78.877, A4 107.384, A5 -59.845, A6 0.000, E1 263.45, E2 0, E3 0, E4 0, E5 0, E6 0} C_DIS
   SPTP {A1 10.261, A2 -63.436, A3 78.786, A4 109.322, A5 -59.110, A6 0.000, E1 262.51, E2 0, E3 0, E4 0, E5 0, E6 0} C_DIS
   SPTP {A1 9.970, A2 -63.873, A3 78.672, A4 111.303, A5 -58.427, A6 0.000, E1 261.52, E2 0, E3 0, E4 0, E5 0, E6 0} C_DIS
   SPTP {A1 9.668, A2 -64.283, A3 78.528, A4 113.327, A5 -57.807, A6 0.000, E1 260.5, E2 0, E3 0, E4 0, E5 0, E6 0} C_DIS
   SPTP {A1 9.358, A2 -64.661, A3 78.350, A4 115.391, A5 -57.263, A6 0.000, E1 259.44, E2 0, E3 0, E4 0, E5 0, E6 0} C_DIS
   SPTP {A1 9.043, A2 -65.103, A3 78.473, A4 116.986, A5 -56.445, A6 0.000, E1 259.2, E2 0, E3 0, E4 0, E5 0, E6 0} C_DIS
   SPTP {A1 8.725, A2 -65.612, A3 78.874, A4 118.169, A5 -55.349, A6 0.000, E1 259.65, E2 0, E3 0, E4 0, E5 0, E6 0} C_DIS
   SPTP {A1 8.405, A2 -66.106, A3 79.272, A4 119.364, A5 -54.271, A6 0.000, E1 260.1, E2 0, E3 0, E4 0, E5 0, E6 0} C_DIS
   SPTP {A1 8.085, A2 -66.582, A3 79.662, A4 120.567, A5 -53.217, A6 0.000, E1 260.55, E2 0, E3 0, E4 0, E5 0, E6 0} C_DIS
   SPTP {A1 7.767, A2 -67.042, A3 80.046, A4 121.777, A5 -52.190, A6 0.000, E1 261, E2 0, E3 0, E4 0, E5 0, E6 0} C_DIS
   SPTP {A1 7.456, A2 -67.528, A3 80.582, A4 122.720, A5 -51.012, A6 0.000, E1 261.85, E2 0, E3 0, E4 0, E5 0, E6 0} C_DIS
   SPTP {A1 7.157, A2 -68.173, A3 81.743, A4 122.571, A5 -49.124, A6 0.000, E1 264.23, E2 0, E3 0, E4 0, E5 0, E6 0} C_DIS
   SPTP {A1 6.866, A2 -68.786, A3 82.888, A4 122.306, A5 -47.249, A6 0.000, E1 266.71, E2 0, E3 0, E4 0, E5 0, E6 0} C_DIS
   SPTP {A1 6.586, A2 -69.365, A3 84.014, A4 121.913, A5 -45.399, A6 0.000, E1 269.31, E2 0, E3 0, E4 0, E5 0, E6 0} C_DIS
   SPTP {A1 6.318, A2 -69.908, A3 85.120, A4 121.376, A5 -43.577, A6 0.000, E1 272.04, E2 0, E3 0, E4 0, E5 0, E6 0} C_DIS
   SPTP {A1 6.066, A2 -70.454, A3 86.396, A4 120.190, A5 -41.574, A6 0.000, E1 275.51, E2 0, E3 0, E4 0, E5 0, E6 0} C_DIS
   SPTP {A1 5.832, A2 -71.042, A3 88.190, A4 117.167, A5 -39.023, A6 0.000, E1 281.09, E2 0, E3 0, E4 0, E5 0, E6 0} C_DIS
   SPTP {A1 5.611, A2 -71.532, A3 89.898, A4 113.573, A5 -36.662, A6 0.000, E1 287.2, E2 0, E3 0, E4 0, E5 0, E6 0} C_DIS
   SPTP {A1 5.403, A2 -71.925, A3 91.517, A4 109.353, A5 -34.533, A6 0.000, E1 293.9, E2 0, E3 0, E4 0, E5 0, E6 0} C_DIS
   SPTP {A1 5.207, A2 -72.219, A3 93.044, A4 104.479, A5 -32.692, A6 0.000, E1 301.22, E2 0, E3 0, E4 0, E5 0, E6 0} C_DIS
   SPTP {A1 5.025, A2 -72.412, A3 94.474, A4 98.963, A5 -31.197, A6 0.000, E1 309.16, E2 0, E3 0, E4 0, E5 0, E6 0} C_DIS
   SPTP {A1 4.854, A2 -72.480, A3 95.928, A4 92.077, A5 -30.139, A6 0.000, E1 318.4, E2 0, E3 0, E4 0, E5 0, E6 0} C_DIS
   SPTP {A1 4.693, A2 -72.402, A3 97.329, A4 84.231, A5 -29.692, A6 0.000, E1 328.55, E2 0, E3 0, E4 0, E5 0, E6 0} C_DIS
   SPTP {A1 4.538, A2 -72.191, A3 98.582, A4 76.311, A5 -29.886, A6 0.000, E1 338.75, E2 0, E3 0, E4 0, E5 0, E6 0} C_DIS
   SPTP {A1 4.389, A2 -71.849, A3 99.682, A4 68.682, A5 -30.701, A6 0.000, E1 348.65, E2 0, E3 0, E4 0, E5 0, E6 0} C_DIS
   SPTP {A1 4.251, A2 -71.378, A3 100.622, A4 61.659, A5 -32.089, A6 0.000, E1 357.93, E2 0, E3 0, E4 0, E5 0, E6 0} C_DIS
   SPTP {A1 4.126, A2 -70.780, A3 101.399, A4 55.426, A5 -33.967, A6 0.000, E1 366.42, E2 0, E3 0, E4 0, E5 0, E6 0} C_DIS
   SPTP {A1 4.012, A2 -70.064, A3 102.010, A4 50.032, A5 -36.235, A6 0.000, E1 374.08, E2 0, E3 0, E4 0, E5 0, E6 0} C_DIS
   SPTP {A1 3.913, A2 -69.233, A3 102.453, A4 45.458, A5 -38.806, A6 0.000, E1 380.93, E2 0, E3 0, E4 0, E5 0, E6 0} C_DIS
   SPTP {A1 3.831, A2 -68.294, A3 102.724, A4 41.640, A5 -41.601, A6 0.000, E1 387.05, E2 0, E3 0, E4 0, E5 0, E6 0} C_DIS
   SPTP {A1 3.767, A2 -67.353, A3 102.839, A4 38.685, A5 -44.308, A6 0.000, E1 392.24, E2 0, E3 0, E4 0, E5 0, E6 0} C_DIS
   SPTP {A1 3.716, A2 -66.610, A3 102.875, A4 36.687, A5 -46.436, A6 0.000, E1 396.26, E2 0, E3 0, E4 0, E5 0, E6 0} C_DIS
   SPTP {A1 3.685, A2 -65.820, A3 102.817, A4 35.000, A5 -48.610, A6 0.000, E1 400.01, E2 0, E3 0, E4 0, E5 0, E6 0} C_DIS
   SPTP {A1 3.674, A2 -64.986, A3 102.665, A4 33.598, A5 -50.815, A6 0.000, E1 403.5, E2 0, E3 0, E4 0, E5 0, E6 0} C_DIS
   SPTP {A1 3.683, A2 -64.113, A3 102.419, A4 32.451, A5 -53.032, A6 0.000, E1 406.77, E2 0, E3 0, E4 0, E5 0, E6 0} C_DIS
   SPTP {A1 3.711, A2 -63.204, A3 102.083, A4 31.530, A5 -55.247, A6 0.000, E1 409.85, E2 0, E3 0, E4 0, E5 0, E6 0} C_DIS
   SPTP {A1 3.757, A2 -62.264, A3 101.656, A4 30.811, A5 -57.447, A6 0.000, E1 412.77, E2 0, E3 0, E4 0, E5 0, E6 0} C_DIS
   SPTP {A1 3.857, A2 -61.672, A3 101.337, A4 30.646, A5 -58.838, A6 0.000, E1 415.13, E2 0, E3 0, E4 0, E5 0, E6 0} C_DIS
   SPTP {A1 3.986, A2 -61.162, A3 101.021, A4 30.695, A5 -60.021, A6 0.000, E1 417.29, E2 0, E3 0, E4 0, E5 0, E6 0} C_DIS
   SPTP {A1 4.130, A2 -60.644, A3 100.666, A4 30.847, A5 -61.191, A6 0.000, E1 419.38, E2 0, E3 0, E4 0, E5 0, E6 0} C_DIS
   SPTP {A1 4.289, A2 -60.117, A3 100.273, A4 31.093, A5 -62.345, A6 0.000, E1 421.4, E2 0, E3 0, E4 0, E5 0, E6 0} C_DIS
   SPTP {A1 4.460, A2 -59.584, A3 99.843, A4 31.419, A5 -63.480, A6 0.000, E1 423.37, E2 0, E3 0, E4 0, E5 0, E6 0} C_DIS
   SPTP {A1 4.642, A2 -59.045, A3 99.375, A4 31.823, A5 -64.594, A6 0.000, E1 425.28, E2 0, E3 0, E4 0, E5 0, E6 0} C_DIS
   SPTP {A1 4.832, A2 -58.501, A3 98.874, A4 32.293, A5 -65.685, A6 0.000, E1 427.14, E2 0, E3 0, E4 0, E5 0, E6 0} C_DIS
   SPTP {A1 5.033, A2 -57.968, A3 98.347, A4 32.839, A5 -66.722, A6 0.000, E1 428.95, E2 0, E3 0, E4 0, E5 0, E6 0} C_DIS
   SPTP {A1 5.306, A2 -57.801, A3 98.022, A4 33.817, A5 -67.040, A6 0.000, E1 430.4, E2 0, E3 0, E4 0, E5 0, E6 0} C_DIS
   SPTP {A1 5.584, A2 -57.631, A3 97.672, A4 34.843, A5 -67.348, A6 0.000, E1 431.81, E2 0, E3 0, E4 0, E5 0, E6 0} C_DIS
   SPTP {A1 5.866, A2 -57.458, A3 97.298, A4 35.912, A5 -67.644, A6 0.000, E1 433.18, E2 0, E3 0, E4 0, E5 0, E6 0} C_DIS
   SPTP {A1 6.151, A2 -57.283, A3 96.901, A4 37.016, A5 -67.930, A6 0.000, E1 434.52, E2 0, E3 0, E4 0, E5 0, E6 0} C_DIS
   SPTP {A1 6.436, A2 -57.104, A3 96.480, A4 38.152, A5 -68.205, A6 0.000, E1 435.82, E2 0, E3 0, E4 0, E5 0, E6 0} C_DIS
   SPTP {A1 6.721, A2 -56.923, A3 96.037, A4 39.314, A5 -68.470, A6 0.000, E1 437.1, E2 0, E3 0, E4 0, E5 0, E6 0} C_DIS
   SPTP {A1 7.005, A2 -56.740, A3 95.572, A4 40.497, A5 -68.724, A6 0.000, E1 438.36, E2 0, E3 0, E4 0, E5 0, E6 0} C_DIS
   SPTP {A1 7.285, A2 -56.555, A3 95.087, A4 41.698, A5 -68.968, A6 0.000, E1 439.59, E2 0, E3 0, E4 0, E5 0, E6 0} C_DIS
   SPTP {A1 7.562, A2 -56.368, A3 94.583, A4 42.912, A5 -69.201, A6 0.000, E1 440.8, E2 0, E3 0, E4 0, E5 0, E6 0} C_DIS
   SPTP {A1 7.834, A2 -56.180, A3 94.060, A4 44.136, A5 -69.422, A6 0.000, E1 442, E2 0, E3 0, E4 0, E5 0, E6 0} C_DIS
   SPTP {A1 8.100, A2 -55.992, A3 93.521, A4 45.367, A5 -69.634, A6 0.000, E1 443.19, E2 0, E3 0, E4 0, E5 0, E6 0} C_DIS
   SPTP {A1 8.364, A2 -55.848, A3 92.998, A4 46.644, A5 -69.759, A6 0.000, E1 444.29, E2 0, E3 0, E4 0, E5 0, E6 0} C_DIS
   SPTP {A1 8.630, A2 -55.783, A3 92.518, A4 48.005, A5 -69.744, A6 0.000, E1 445.26, E2 0, E3 0, E4 0, E5 0, E6 0} C_DIS
   SPTP {A1 8.888, A2 -55.716, A3 92.022, A4 49.368, A5 -69.724, A6 0.000, E1 446.21, E2 0, E3 0, E4 0, E5 0, E6 0} C_DIS
   SPTP {A1 9.137, A2 -55.647, A3 91.511, A4 50.733, A5 -69.701, A6 0.000, E1 447.16, E2 0, E3 0, E4 0, E5 0, E6 0} C_DIS
   SPTP {A1 9.378, A2 -55.578, A3 90.989, A4 52.095, A5 -69.671, A6 0.000, E1 448.09, E2 0, E3 0, E4 0, E5 0, E6 0} C_DIS
   SPTP {A1 9.610, A2 -55.508, A3 90.456, A4 53.453, A5 -69.637, A6 0.000, E1 449.01, E2 0, E3 0, E4 0, E5 0, E6 0} C_DIS
   SPTP {A1 9.832, A2 -55.440, A3 89.914, A4 54.803, A5 -69.596, A6 0.000, E1 449.94, E2 0, E3 0, E4 0, E5 0, E6 0} C_DIS
   SPTP {A1 10.044, A2 -55.374, A3 89.366, A4 56.146, A5 -69.550, A6 0.000, E1 450.85, E2 0, E3 0, E4 0, E5 0, E6 0} C_DIS
   SPTP {A1 10.245, A2 -55.311, A3 88.815, A4 57.475, A5 -69.494, A6 0.000, E1 451.77, E2 0, E3 0, E4 0, E5 0, E6 0} C_DIS
   SPTP {A1 10.436, A2 -55.251, A3 88.262, A4 58.794, A5 -69.432, A6 0.000, E1 452.69, E2 0, E3 0, E4 0, E5 0, E6 0} C_DIS
   SPTP {A1 10.613, A2 -55.198, A3 87.717, A4 60.081, A5 -69.364, A6 0.000, E1 453.61, E2 0, E3 0, E4 0, E5 0, E6 0} C_DIS
   SPTP {A1 10.769, A2 -55.152, A3 87.200, A4 61.302, A5 -69.304, A6 0.000, E1 454.51, E2 0, E3 0, E4 0, E5 0, E6 0} C_DIS
   SPTP {A1 10.903, A2 -55.113, A3 86.718, A4 62.441, A5 -69.255, A6 0.000, E1 455.39, E2 0, E3 0, E4 0, E5 0, E6 0} C_DIS
   SPTP {A1 11.011, A2 -55.083, A3 86.286, A4 63.474, A5 -69.226, A6 0.000, E1 456.25, E2 0, E3 0, E4 0, E5 0, E6 0} C_DIS
   SPTP {A1 11.112, A2 -55.062, A3 85.864, A4 64.490, A5 -69.183, A6 0.000, E1 457.13, E2 0, E3 0, E4 0, E5 0, E6 0} C_DIS
   SPTP {A1 11.204, A2 -55.050, A3 85.454, A4 65.487, A5 -69.126, A6 0.000, E1 458.01, E2 0, E3 0, E4 0, E5 0, E6 0} C_DIS
   SPTP {A1 11.287, A2 -55.053, A3 85.063, A4 66.461, A5 -69.048, A6 0.000, E1 458.91, E2 0, E3 0, E4 0, E5 0, E6 0} C_DIS
   SPTP {A1 11.362, A2 -55.066, A3 84.687, A4 67.417, A5 -68.953, A6 0.000, E1 459.83, E2 0, E3 0, E4 0, E5 0, E6 0} C_DIS
   SPTP {A1 11.428, A2 -55.093, A3 84.330, A4 68.352, A5 -68.839, A6 0.000, E1 460.76, E2 0, E3 0, E4 0, E5 0, E6 0} C_DIS
   SPTP {A1 11.487, A2 -55.133, A3 83.993, A4 69.266, A5 -68.704, A6 0.000, E1 461.7, E2 0, E3 0, E4 0, E5 0, E6 0} C_DIS
   SPTP {A1 11.537, A2 -55.188, A3 83.678, A4 70.159, A5 -68.547, A6 0.000, E1 462.66, E2 0, E3 0, E4 0, E5 0, E6 0} C_DIS
   SPTP {A1 11.579, A2 -55.258, A3 83.386, A4 71.032, A5 -68.370, A6 0.000, E1 463.64, E2 0, E3 0, E4 0, E5 0, E6 0} C_DIS
   SPTP {A1 11.612, A2 -55.343, A3 83.119, A4 71.882, A5 -68.166, A6 0.000, E1 464.63, E2 0, E3 0, E4 0, E5 0, E6 0} C_DIS
   SPTP {A1 11.638, A2 -55.446, A3 82.878, A4 72.711, A5 -67.937, A6 0.000, E1 465.64, E2 0, E3 0, E4 0, E5 0, E6 0} C_DIS
   SPTP {A1 11.655, A2 -55.566, A3 82.664, A4 73.517, A5 -67.682, A6 0.000, E1 466.67, E2 0, E3 0, E4 0, E5 0, E6 0} C_DIS
   SPTP {A1 11.664, A2 -55.703, A3 82.478, A4 74.302, A5 -67.399, A6 0.000, E1 467.71, E2 0, E3 0, E4 0, E5 0, E6 0} C_DIS
   SPTP {A1 11.666, A2 -55.857, A3 82.321, A4 75.066, A5 -67.090, A6 0.000, E1 468.77, E2 0, E3 0, E4 0, E5 0, E6 0} C_DIS
   SPTP {A1 11.659, A2 -56.029, A3 82.192, A4 75.808, A5 -66.751, A6 0.000, E1 469.85, E2 0, E3 0, E4 0, E5 0, E6 0} C_DIS
   SPTP {A1 11.645, A2 -56.218, A3 82.093, A4 76.529, A5 -66.384, A6 0.000, E1 470.94, E2 0, E3 0, E4 0, E5 0, E6 0} C_DIS
   SPTP {A1 11.618, A2 -56.450, A3 82.052, A4 77.247, A5 -65.972, A6 0.000, E1 471.89, E2 0, E3 0, E4 0, E5 0, E6 0} C_DIS
   SPTP {A1 11.580, A2 -56.725, A3 82.069, A4 77.967, A5 -65.516, A6 0.000, E1 472.68, E2 0, E3 0, E4 0, E5 0, E6 0} C_DIS
   SPTP {A1 11.534, A2 -57.012, A3 82.106, A4 78.673, A5 -65.038, A6 0.000, E1 473.49, E2 0, E3 0, E4 0, E5 0, E6 0} C_DIS
   SPTP {A1 11.481, A2 -57.312, A3 82.165, A4 79.364, A5 -64.535, A6 0.000, E1 474.29, E2 0, E3 0, E4 0, E5 0, E6 0} C_DIS
   SPTP {A1 11.420, A2 -57.627, A3 82.247, A4 80.040, A5 -64.003, A6 0.000, E1 475.11, E2 0, E3 0, E4 0, E5 0, E6 0} C_DIS
   SPTP {A1 11.352, A2 -57.953, A3 82.350, A4 80.701, A5 -63.446, A6 0.000, E1 475.93, E2 0, E3 0, E4 0, E5 0, E6 0} C_DIS
   SPTP {A1 11.276, A2 -58.293, A3 82.475, A4 81.348, A5 -62.862, A6 0.000, E1 476.76, E2 0, E3 0, E4 0, E5 0, E6 0} C_DIS
   SPTP {A1 11.192, A2 -58.645, A3 82.622, A4 81.981, A5 -62.250, A6 0.000, E1 477.59, E2 0, E3 0, E4 0, E5 0, E6 0} C_DIS
   SPTP {A1 11.100, A2 -59.010, A3 82.791, A4 82.598, A5 -61.610, A6 0.000, E1 478.43, E2 0, E3 0, E4 0, E5 0, E6 0} C_DIS
   SPTP {A1 10.999, A2 -59.386, A3 82.980, A4 83.203, A5 -60.942, A6 0.000, E1 479.28, E2 0, E3 0, E4 0, E5 0, E6 0} C_DIS
   SPTP {A1 10.890, A2 -59.773, A3 83.189, A4 83.793, A5 -60.245, A6 0.000, E1 480.12, E2 0, E3 0, E4 0, E5 0, E6 0} C_DIS
   SPTP {A1 10.773, A2 -60.172, A3 83.418, A4 84.370, A5 -59.520, A6 0.000, E1 480.97, E2 0, E3 0, E4 0, E5 0, E6 0} C_DIS
   SPTP {A1 10.652, A2 -60.623, A3 83.591, A4 85.284, A5 -58.680, A6 0.000, E1 481.42, E2 0, E3 0, E4 0, E5 0, E6 0} C_DIS
   SPTP {A1 10.523, A2 -61.099, A3 83.733, A4 86.390, A5 -57.778, A6 0.000, E1 481.65, E2 0, E3 0, E4 0, E5 0, E6 0} C_DIS
   SPTP {A1 10.383, A2 -61.577, A3 83.878, A4 87.510, A5 -56.864, A6 0.000, E1 481.85, E2 0, E3 0, E4 0, E5 0, E6 0} C_DIS
   SPTP {A1 10.231, A2 -62.057, A3 84.030, A4 88.642, A5 -55.934, A6 0.000, E1 482.03, E2 0, E3 0, E4 0, E5 0, E6 0} C_DIS
   SPTP {A1 10.067, A2 -62.539, A3 84.187, A4 89.790, A5 -54.990, A6 0.000, E1 482.17, E2 0, E3 0, E4 0, E5 0, E6 0} C_DIS
   SPTP {A1 9.891, A2 -63.020, A3 84.347, A4 90.956, A5 -54.035, A6 0.000, E1 482.29, E2 0, E3 0, E4 0, E5 0, E6 0} C_DIS
   SPTP {A1 9.704, A2 -63.501, A3 84.511, A4 92.143, A5 -53.069, A6 0.000, E1 482.37, E2 0, E3 0, E4 0, E5 0, E6 0} C_DIS
   SPTP {A1 9.504, A2 -63.982, A3 84.678, A4 93.352, A5 -52.091, A6 0.000, E1 482.41, E2 0, E3 0, E4 0, E5 0, E6 0} C_DIS
   SPTP {A1 9.292, A2 -64.461, A3 84.848, A4 94.587, A5 -51.102, A6 0.000, E1 482.42, E2 0, E3 0, E4 0, E5 0, E6 0} C_DIS
   SPTP {A1 9.067, A2 -64.938, A3 85.019, A4 95.850, A5 -50.104, A6 0.000, E1 482.39, E2 0, E3 0, E4 0, E5 0, E6 0} C_DIS
   SPTP {A1 8.831, A2 -65.412, A3 85.192, A4 97.145, A5 -49.100, A6 0.000, E1 482.31, E2 0, E3 0, E4 0, E5 0, E6 0} C_DIS
   SPTP {A1 8.583, A2 -65.882, A3 85.365, A4 98.475, A5 -48.089, A6 0.000, E1 482.19, E2 0, E3 0, E4 0, E5 0, E6 0} C_DIS
   SPTP {A1 8.322, A2 -66.349, A3 85.539, A4 99.843, A5 -47.073, A6 0.000, E1 482.02, E2 0, E3 0, E4 0, E5 0, E6 0} C_DIS
   SPTP {A1 8.050, A2 -66.811, A3 85.712, A4 101.253, A5 -46.055, A6 0.000, E1 481.79, E2 0, E3 0, E4 0, E5 0, E6 0} C_DIS
   SPTP {A1 7.766, A2 -67.265, A3 85.881, A4 102.711, A5 -45.039, A6 0.000, E1 481.51, E2 0, E3 0, E4 0, E5 0, E6 0} C_DIS
   SPTP {A1 7.455, A2 -67.725, A3 85.951, A4 104.660, A5 -43.950, A6 0.000, E1 480.94, E2 0, E3 0, E4 0, E5 0, E6 0} C_DIS
   SPTP {A1 7.129, A2 -68.174, A3 86.006, A4 106.725, A5 -42.874, A6 0.000, E1 480.26, E2 0, E3 0, E4 0, E5 0, E6 0} C_DIS
   SPTP {A1 6.788, A2 -68.612, A3 86.058, A4 108.873, A5 -41.818, A6 0.000, E1 479.49, E2 0, E3 0, E4 0, E5 0, E6 0} C_DIS
   SPTP {A1 6.432, A2 -69.039, A3 86.107, A4 111.107, A5 -40.787, A6 0.000, E1 478.63, E2 0, E3 0, E4 0, E5 0, E6 0} C_DIS
   SPTP {A1 6.063, A2 -69.452, A3 86.150, A4 113.433, A5 -39.785, A6 0.000, E1 477.66, E2 0, E3 0, E4 0, E5 0, E6 0} C_DIS
   SPTP {A1 5.681, A2 -69.852, A3 86.189, A4 115.854, A5 -38.819, A6 0.000, E1 476.6, E2 0, E3 0, E4 0, E5 0, E6 0} C_DIS
   SPTP {A1 5.288, A2 -70.236, A3 86.222, A4 118.372, A5 -37.897, A6 0.000, E1 475.44, E2 0, E3 0, E4 0, E5 0, E6 0} C_DIS
   SPTP {A1 4.885, A2 -70.605, A3 86.248, A4 120.987, A5 -37.024, A6 0.000, E1 474.19, E2 0, E3 0, E4 0, E5 0, E6 0} C_DIS
   SPTP {A1 4.473, A2 -70.957, A3 86.267, A4 123.698, A5 -36.208, A6 0.000, E1 472.83, E2 0, E3 0, E4 0, E5 0, E6 0} C_DIS
   SPTP {A1 4.053, A2 -71.292, A3 86.279, A4 126.500, A5 -35.454, A6 0.000, E1 471.4, E2 0, E3 0, E4 0, E5 0, E6 0} C_DIS
   SPTP {A1 3.628, A2 -71.610, A3 86.284, A4 129.387, A5 -34.768, A6 0.000, E1 469.88, E2 0, E3 0, E4 0, E5 0, E6 0} C_DIS
   SPTP {A1 3.197, A2 -71.912, A3 86.284, A4 132.350, A5 -34.150, A6 0.000, E1 468.29, E2 0, E3 0, E4 0, E5 0, E6 0} C_DIS
   SPTP {A1 2.765, A2 -72.196, A3 86.276, A4 135.372, A5 -33.613, A6 0.000, E1 466.66, E2 0, E3 0, E4 0, E5 0, E6 0} C_DIS
   SPTP {A1 2.331, A2 -72.498, A3 86.397, A4 138.157, A5 -32.944, A6 0.000, E1 465.35, E2 0, E3 0, E4 0, E5 0, E6 0} C_DIS
   SPTP {A1 1.896, A2 -72.873, A3 86.838, A4 140.350, A5 -31.812, A6 0.000, E1 464.78, E2 0, E3 0, E4 0, E5 0, E6 0} C_DIS
   SPTP {A1 1.464, A2 -73.235, A3 87.285, A4 142.618, A5 -30.704, A6 0.000, E1 464.14, E2 0, E3 0, E4 0, E5 0, E6 0} C_DIS
   SPTP {A1 1.038, A2 -73.586, A3 87.739, A4 144.959, A5 -29.625, A6 0.000, E1 463.44, E2 0, E3 0, E4 0, E5 0, E6 0} C_DIS
   SPTP {A1 0.621, A2 -73.924, A3 88.198, A4 147.357, A5 -28.581, A6 0.000, E1 462.7, E2 0, E3 0, E4 0, E5 0, E6 0} C_DIS
   SPTP {A1 0.218, A2 -74.251, A3 88.664, A4 149.797, A5 -27.575, A6 0.000, E1 461.92, E2 0, E3 0, E4 0, E5 0, E6 0} C_DIS
   SPTP {A1 -0.168, A2 -74.567, A3 89.137, A4 152.259, A5 -26.608, A6 0.000, E1 461.16, E2 0, E3 0, E4 0, E5 0, E6 0} C_DIS
   SPTP {A1 -0.529, A2 -74.887, A3 89.681, A4 154.567, A5 -25.563, A6 0.000, E1 460.57, E2 0, E3 0, E4 0, E5 0, E6 0} C_DIS
   SPTP {A1 -0.852, A2 -75.337, A3 90.882, A4 155.363, A5 -23.306, A6 0.000, E1 461.51, E2 0, E3 0, E4 0, E5 0, E6 0} C_DIS
   SPTP {A1 -1.145, A2 -75.752, A3 92.068, A4 156.033, A5 -21.048, A6 0.000, E1 462.59, E2 0, E3 0, E4 0, E5 0, E6 0} C_DIS
   SPTP {A1 -1.403, A2 -76.132, A3 93.234, A4 156.476, A5 -18.799, A6 0.000, E1 463.91, E2 0, E3 0, E4 0, E5 0, E6 0} C_DIS
   SPTP {A1 -1.616, A2 -76.476, A3 94.381, A4 156.531, A5 -16.567, A6 0.000, E1 465.65, E2 0, E3 0, E4 0, E5 0, E6 0} C_DIS
   SPTP {A1 -1.780, A2 -76.791, A3 95.585, A4 155.636, A5 -14.185, A6 0.000, E1 468.36, E2 0, E3 0, E4 0, E5 0, E6 0} C_DIS
   SPTP {A1 -1.891, A2 -77.087, A3 97.449, A4 148.824, A5 -10.278, A6 0.000, E1 476.94, E2 0, E3 0, E4 0, E5 0, E6 0} C_DIS
   SPTP {A1 -1.953, A2 -77.255, A3 99.196, A4 133.046, A5 -6.784, A6 0.000, E1 494.49, E2 0, E3 0, E4 0, E5 0, E6 0} C_DIS
   SPTP {A1 -1.964, A2 -77.292, A3 100.819, A4 95.300, A5 -4.787, A6 0.000, E1 534.02, E2 0, E3 0, E4 0, E5 0, E6 0} C_DIS
   SPTP {A1 -1.918, A2 -77.196, A3 102.311, A4 51.746, A5 -6.079, A6 0.000, E1 579.37, E2 0, E3 0, E4 0, E5 0, E6 0} C_DIS
   SPTP {A1 -1.834, A2 -76.787, A3 104.036, A4 27.490, A5 -10.708, A6 0.000, E1 605.44, E2 0, E3 0, E4 0, E5 0, E6 0} C_DIS
   SPTP {A1 -1.707, A2 -76.005, A3 105.644, A4 18.371, A5 -16.863, A6 0.000, E1 616.37, E2 0, E3 0, E4 0, E5 0, E6 0} C_DIS
   SPTP {A1 -1.547, A2 -74.924, A3 106.893, A4 14.620, A5 -23.206, A6 0.000, E1 621.94, E2 0, E3 0, E4 0, E5 0, E6 0} C_DIS
   SPTP {A1 -1.368, A2 -73.404, A3 107.816, A4 12.511, A5 -30.130, A6 0.000, E1 625.93, E2 0, E3 0, E4 0, E5 0, E6 0} C_DIS
   SPTP {A1 -1.172, A2 -71.060, A3 108.277, A4 10.977, A5 -38.534, A6 0.000, E1 629.59, E2 0, E3 0, E4 0, E5 0, E6 0} C_DIS
   SPTP {A1 -0.977, A2 -68.314, A3 108.033, A4 10.225, A5 -46.680, A6 0.000, E1 632.48, E2 0, E3 0, E4 0, E5 0, E6 0} C_DIS
   SPTP {A1 -0.787, A2 -65.244, A3 107.083, A4 9.903, A5 -54.467, A6 0.000, E1 634.96, E2 0, E3 0, E4 0, E5 0, E6 0} C_DIS
   SPTP {A1 -0.567, A2 -62.087, A3 105.527, A4 9.944, A5 -61.490, A6 0.000, E1 637.29, E2 0, E3 0, E4 0, E5 0, E6 0} C_DIS
   SPTP {A1 -0.160, A2 -59.418, A3 103.791, A4 10.710, A5 -66.845, A6 0.000, E1 639.7, E2 0, E3 0, E4 0, E5 0, E6 0} C_DIS
   SPTP {A1 0.263, A2 -56.693, A3 101.652, A4 11.628, A5 -71.832, A6 0.000, E1 642.07, E2 0, E3 0, E4 0, E5 0, E6 0} C_DIS
   SPTP {A1 0.701, A2 -53.940, A3 99.129, A4 12.698, A5 -76.439, A6 0.000, E1 644.39, E2 0, E3 0, E4 0, E5 0, E6 0} C_DIS
   SPTP {A1 1.148, A2 -51.181, A3 96.240, A4 13.905, A5 -80.657, A6 0.000, E1 646.68, E2 0, E3 0, E4 0, E5 0, E6 0} C_DIS
   SPTP {A1 1.601, A2 -48.430, A3 93.005, A4 15.231, A5 -84.487, A6 0.000, E1 648.95, E2 0, E3 0, E4 0, E5 0, E6 0} C_DIS
   SPTP {A1 2.058, A2 -45.691, A3 89.430, A4 16.683, A5 -87.935, A6 0.000, E1 651.19, E2 0, E3 0, E4 0, E5 0, E6 0} C_DIS
   SPTP {A1 2.522, A2 -42.956, A3 85.510, A4 18.273, A5 -91.012, A6 0.000, E1 653.37, E2 0, E3 0, E4 0, E5 0, E6 0} C_DIS
   SPTP {A1 2.985, A2 -40.216, A3 81.243, A4 19.977, A5 -93.726, A6 0.000, E1 655.48, E2 0, E3 0, E4 0, E5 0, E6 0} C_DIS
   SPTP {A1 3.446, A2 -37.448, A3 76.601, A4 21.790, A5 -96.086, A6 0.000, E1 657.49, E2 0, E3 0, E4 0, E5 0, E6 0} C_DIS
   SPTP {A1 3.911, A2 -34.865, A3 71.950, A4 23.714, A5 -97.923, A6 0.000, E1 659.32, E2 0, E3 0, E4 0, E5 0, E6 0} C_DIS
   SPTP {A1 4.479, A2 -34.761, A3 71.245, A4 25.892, A5 -97.840, A6 0.000, E1 660.62, E2 0, E3 0, E4 0, E5 0, E6 0} C_DIS
   SPTP {A1 5.040, A2 -34.638, A3 70.452, A4 28.139, A5 -97.723, A6 0.000, E1 661.75, E2 0, E3 0, E4 0, E5 0, E6 0} C_DIS
   SPTP {A1 5.590, A2 -34.492, A3 69.566, A4 30.437, A5 -97.578, A6 0.000, E1 662.74, E2 0, E3 0, E4 0, E5 0, E6 0} C_DIS
   SPTP {A1 6.104, A2 -34.707, A3 69.281, A4 32.662, A5 -97.185, A6 0.000, E1 663.45, E2 0, E3 0, E4 0, E5 0, E6 0} C_DIS
   SPTP {A1 6.581, A2 -35.355, A3 69.727, A4 34.796, A5 -96.500, A6 0.000, E1 663.83, E2 0, E3 0, E4 0, E5 0, E6 0} C_DIS
   SPTP {A1 7.012, A2 -35.910, A3 70.027, A4 36.787, A5 -95.860, A6 0.000, E1 664.07, E2 0, E3 0, E4 0, E5 0, E6 0} C_DIS
   SPTP {A1 7.434, A2 -36.432, A3 70.237, A4 38.796, A5 -95.213, A6 0.000, E1 664.23, E2 0, E3 0, E4 0, E5 0, E6 0} C_DIS
   SPTP {A1 7.434, A2 -36.418, A3 70.220, A4 38.809, A5 -95.225, A6 0.000, E1 664.21, E2 0, E3 0, E4 0, E5 0, E6 0} C_DIS
   SPTP {A1 7.882, A2 -36.955, A3 70.361, A4 41.005, A5 -94.514, A6 0.000, E1 664.31, E2 0, E3 0, E4 0, E5 0, E6 0} C_DIS
   SPTP {A1 8.285, A2 -37.739, A3 70.924, A4 43.063, A5 -93.633, A6 0.000, E1 664.17, E2 0, E3 0, E4 0, E5 0, E6 0} C_DIS
   SPTP {A1 8.648, A2 -38.761, A3 71.883, A4 44.999, A5 -92.568, A6 0.000, E1 663.75, E2 0, E3 0, E4 0, E5 0, E6 0} C_DIS
   SPTP {A1 9.003, A2 -39.745, A3 72.728, A4 46.956, A5 -91.486, A6 0.000, E1 663.25, E2 0, E3 0, E4 0, E5 0, E6 0} C_DIS
   SPTP {A1 9.351, A2 -40.697, A3 73.472, A4 48.934, A5 -90.388, A6 0.000, E1 662.69, E2 0, E3 0, E4 0, E5 0, E6 0} C_DIS
   SPTP {A1 9.688, A2 -41.625, A3 74.133, A4 50.923, A5 -89.277, A6 0.000, E1 662.06, E2 0, E3 0, E4 0, E5 0, E6 0} C_DIS
   SPTP {A1 10.013, A2 -42.535, A3 74.723, A4 52.920, A5 -88.149, A6 0.000, E1 661.4, E2 0, E3 0, E4 0, E5 0, E6 0} C_DIS
   SPTP {A1 10.324, A2 -43.432, A3 75.253, A4 54.921, A5 -87.004, A6 0.000, E1 660.68, E2 0, E3 0, E4 0, E5 0, E6 0} C_DIS
   SPTP {A1 10.620, A2 -44.319, A3 75.730, A4 56.923, A5 -85.843, A6 0.000, E1 659.93, E2 0, E3 0, E4 0, E5 0, E6 0} C_DIS
   SPTP {A1 10.875, A2 -45.310, A3 76.374, A4 58.825, A5 -84.599, A6 0.000, E1 658.96, E2 0, E3 0, E4 0, E5 0, E6 0} C_DIS
   SPTP {A1 11.105, A2 -46.337, A3 77.045, A4 60.697, A5 -83.304, A6 0.000, E1 657.87, E2 0, E3 0, E4 0, E5 0, E6 0} C_DIS
   SPTP {A1 11.321, A2 -47.333, A3 77.629, A4 62.607, A5 -82.018, A6 0.000, E1 656.69, E2 0, E3 0, E4 0, E5 0, E6 0} C_DIS
   SPTP {A1 11.518, A2 -48.323, A3 78.163, A4 64.530, A5 -80.714, A6 0.000, E1 655.46, E2 0, E3 0, E4 0, E5 0, E6 0} C_DIS
   SPTP {A1 11.698, A2 -49.294, A3 78.632, A4 66.483, A5 -79.412, A6 0.000, E1 654.16, E2 0, E3 0, E4 0, E5 0, E6 0} C_DIS
   SPTP {A1 11.856, A2 -50.256, A3 79.055, A4 68.456, A5 -78.101, A6 0.000, E1 652.79, E2 0, E3 0, E4 0, E5 0, E6 0} C_DIS
   SPTP {A1 11.993, A2 -51.204, A3 79.425, A4 70.458, A5 -76.791, A6 0.000, E1 651.36, E2 0, E3 0, E4 0, E5 0, E6 0} C_DIS
   SPTP {A1 12.107, A2 -52.133, A3 79.736, A4 72.498, A5 -75.492, A6 0.000, E1 649.85, E2 0, E3 0, E4 0, E5 0, E6 0} C_DIS
   SPTP {A1 12.197, A2 -53.050, A3 80.001, A4 74.571, A5 -74.198, A6 0.000, E1 648.26, E2 0, E3 0, E4 0, E5 0, E6 0} C_DIS
   SPTP {A1 12.263, A2 -53.939, A3 80.199, A4 76.696, A5 -72.933, A6 0.000, E1 646.57, E2 0, E3 0, E4 0, E5 0, E6 0} C_DIS
   SPTP {A1 12.303, A2 -54.815, A3 80.354, A4 78.862, A5 -71.681, A6 0.000, E1 644.81, E2 0, E3 0, E4 0, E5 0, E6 0} C_DIS
   SPTP {A1 12.319, A2 -55.652, A3 80.430, A4 81.094, A5 -70.482, A6 0.000, E1 642.94, E2 0, E3 0, E4 0, E5 0, E6 0} C_DIS
   SPTP {A1 12.306, A2 -56.471, A3 80.461, A4 83.375, A5 -69.310, A6 0.000, E1 640.98, E2 0, E3 0, E4 0, E5 0, E6 0} C_DIS
   SPTP {A1 12.267, A2 -57.235, A3 80.419, A4 85.682, A5 -68.219, A6 0.000, E1 638.99, E2 0, E3 0, E4 0, E5 0, E6 0} C_DIS
   SPTP {A1 12.198, A2 -57.917, A3 80.368, A4 87.770, A5 -67.210, A6 0.000, E1 637.48, E2 0, E3 0, E4 0, E5 0, E6 0} C_DIS
   SPTP {A1 12.104, A2 -58.576, A3 80.287, A4 89.884, A5 -66.235, A6 0.000, E1 635.95, E2 0, E3 0, E4 0, E5 0, E6 0} C_DIS
   SPTP {A1 11.986, A2 -59.216, A3 80.176, A4 92.045, A5 -65.294, A6 0.000, E1 634.34, E2 0, E3 0, E4 0, E5 0, E6 0} C_DIS
   SPTP {A1 11.845, A2 -59.834, A3 80.028, A4 94.257, A5 -64.396, A6 0.000, E1 632.64, E2 0, E3 0, E4 0, E5 0, E6 0} C_DIS
   SPTP {A1 11.680, A2 -60.423, A3 79.838, A4 96.527, A5 -63.554, A6 0.000, E1 630.87, E2 0, E3 0, E4 0, E5 0, E6 0} C_DIS
   SPTP {A1 11.493, A2 -60.982, A3 79.604, A4 98.853, A5 -62.775, A6 0.000, E1 629.02, E2 0, E3 0, E4 0, E5 0, E6 0} C_DIS
   SPTP {A1 11.284, A2 -61.503, A3 79.316, A4 101.240, A5 -62.078, A6 0.000, E1 627.09, E2 0, E3 0, E4 0, E5 0, E6 0} C_DIS
   SPTP {A1 11.056, A2 -61.985, A3 78.999, A4 103.626, A5 -61.451, A6 0.000, E1 625.21, E2 0, E3 0, E4 0, E5 0, E6 0} C_DIS
   SPTP {A1 10.810, A2 -62.476, A3 78.935, A4 105.480, A5 -60.656, A6 0.000, E1 624.37, E2 0, E3 0, E4 0, E5 0, E6 0} C_DIS
   SPTP {A1 10.548, A2 -62.955, A3 78.862, A4 107.373, A5 -59.883, A6 0.000, E1 623.47, E2 0, E3 0, E4 0, E5 0, E6 0} C_DIS
   SPTP {A1 10.269, A2 -63.417, A3 78.774, A4 109.308, A5 -59.145, A6 0.000, E1 622.53, E2 0, E3 0, E4 0, E5 0, E6 0} C_DIS
   SPTP {A1 9.978, A2 -63.856, A3 78.663, A4 111.286, A5 -58.458, A6 0.000, E1 621.55, E2 0, E3 0, E4 0, E5 0, E6 0} C_DIS
   SPTP {A1 9.676, A2 -64.268, A3 78.521, A4 113.307, A5 -57.835, A6 0.000, E1 620.52, E2 0, E3 0, E4 0, E5 0, E6 0} C_DIS
   SPTP {A1 9.365, A2 -64.647, A3 78.346, A4 115.369, A5 -57.287, A6 0.000, E1 619.46, E2 0, E3 0, E4 0, E5 0, E6 0} C_DIS
   SPTP {A1 9.050, A2 -65.090, A3 78.465, A4 116.970, A5 -56.472, A6 0.000, E1 619.21, E2 0, E3 0, E4 0, E5 0, E6 0} C_DIS
   SPTP {A1 8.731, A2 -65.600, A3 78.869, A4 118.152, A5 -55.372, A6 0.000, E1 619.66, E2 0, E3 0, E4 0, E5 0, E6 0} C_DIS
   SPTP {A1 8.410, A2 -66.096, A3 79.269, A4 119.345, A5 -54.290, A6 0.000, E1 620.11, E2 0, E3 0, E4 0, E5 0, E6 0} C_DIS
   SPTP {A1 8.090, A2 -66.574, A3 79.662, A4 120.547, A5 -53.232, A6 0.000, E1 620.55, E2 0, E3 0, E4 0, E5 0, E6 0} C_DIS
   SPTP {A1 7.771, A2 -67.035, A3 80.048, A4 121.756, A5 -52.201, A6 0.000, E1 621, E2 0, E3 0, E4 0, E5 0, E6 0} C_DIS
   SPTP {A1 7.460, A2 -67.519, A3 80.575, A4 122.716, A5 -51.033, A6 0.000, E1 621.82, E2 0, E3 0, E4 0, E5 0, E6 0} C_DIS
   SPTP {A1 7.160, A2 -68.166, A3 81.737, A4 122.569, A5 -49.142, A6 0.000, E1 624.2, E2 0, E3 0, E4 0, E5 0, E6 0} C_DIS
   SPTP {A1 6.868, A2 -68.780, A3 82.883, A4 122.307, A5 -47.264, A6 0.000, E1 626.67, E2 0, E3 0, E4 0, E5 0, E6 0} C_DIS
   SPTP {A1 6.587, A2 -69.360, A3 84.009, A4 121.917, A5 -45.411, A6 0.000, E1 629.26, E2 0, E3 0, E4 0, E5 0, E6 0} C_DIS
   SPTP {A1 6.318, A2 -69.905, A3 85.116, A4 121.384, A5 -43.586, A6 0.000, E1 631.98, E2 0, E3 0, E4 0, E5 0, E6 0} C_DIS
   SPTP {A1 6.065, A2 -70.449, A3 86.378, A4 120.240, A5 -41.597, A6 0.000, E1 635.4, E2 0, E3 0, E4 0, E5 0, E6 0} C_DIS
   SPTP {A1 5.829, A2 -71.038, A3 88.172, A4 117.231, A5 -39.042, A6 0.000, E1 640.96, E2 0, E3 0, E4 0, E5 0, E6 0} C_DIS
   SPTP {A1 5.607, A2 -71.531, A3 89.879, A4 113.652, A5 -36.676, A6 0.000, E1 647.06, E2 0, E3 0, E4 0, E5 0, E6 0} C_DIS
   SPTP {A1 5.398, A2 -71.925, A3 91.499, A4 109.449, A5 -34.541, A6 0.000, E1 653.74, E2 0, E3 0, E4 0, E5 0, E6 0} C_DIS
   SPTP {A1 5.201, A2 -72.222, A3 93.027, A4 104.591, A5 -32.691, A6 0.000, E1 661.04, E2 0, E3 0, E4 0, E5 0, E6 0} C_DIS
   SPTP {A1 5.017, A2 -72.418, A3 94.458, A4 99.089, A5 -31.186, A6 0.000, E1 668.95, E2 0, E3 0, E4 0, E5 0, E6 0} C_DIS
   SPTP {A1 4.846, A2 -72.489, A3 95.907, A4 92.251, A5 -30.115, A6 0.000, E1 678.14, E2 0, E3 0, E4 0, E5 0, E6 0} C_DIS
   SPTP {A1 4.684, A2 -72.415, A3 97.310, A4 84.410, A5 -29.651, A6 0.000, E1 688.29, E2 0, E3 0, E4 0, E5 0, E6 0} C_DIS
   SPTP {A1 4.529, A2 -72.208, A3 98.565, A4 76.485, A5 -29.828, A6 0.000, E1 698.49, E2 0, E3 0, E4 0, E5 0, E6 0} C_DIS
   SPTP {A1 4.380, A2 -71.870, A3 99.668, A4 68.843, A5 -30.627, A6 0.000, E1 708.4, E2 0, E3 0, E4 0, E5 0, E6 0} C_DIS
   SPTP {A1 4.242, A2 -71.403, A3 100.613, A4 61.799, A5 -31.999, A6 0.000, E1 717.7, E2 0, E3 0, E4 0, E5 0, E6 0} C_DIS
   SPTP {A1 4.116, A2 -70.810, A3 101.393, A4 55.545, A5 -33.864, A6 0.000, E1 726.21, E2 0, E3 0, E4 0, E5 0, E6 0} C_DIS
   SPTP {A1 4.003, A2 -70.098, A3 102.008, A4 50.132, A5 -36.122, A6 0.000, E1 733.88, E2 0, E3 0, E4 0, E5 0, E6 0} C_DIS
   SPTP {A1 3.904, A2 -69.271, A3 102.456, A4 45.540, A5 -38.684, A6 0.000, E1 740.75, E2 0, E3 0, E4 0, E5 0, E6 0} C_DIS
   SPTP {A1 3.822, A2 -68.337, A3 102.733, A4 41.704, A5 -41.473, A6 0.000, E1 746.88, E2 0, E3 0, E4 0, E5 0, E6 0} C_DIS
   SPTP {A1 3.758, A2 -67.386, A3 102.850, A4 38.708, A5 -44.210, A6 0.000, E1 752.13, E2 0, E3 0, E4 0, E5 0, E6 0} C_DIS
   SPTP {A1 3.707, A2 -66.645, A3 102.890, A4 36.703, A5 -46.335, A6 0.000, E1 756.15, E2 0, E3 0, E4 0, E5 0, E6 0} C_DIS
   SPTP {A1 3.676, A2 -65.857, A3 102.835, A4 35.011, A5 -48.508, A6 0.000, E1 759.9, E2 0, E3 0, E4 0, E5 0, E6 0} C_DIS
   SPTP {A1 3.666, A2 -65.025, A3 102.686, A4 33.607, A5 -50.712, A6 0.000, E1 763.39, E2 0, E3 0, E4 0, E5 0, E6 0} C_DIS
   SPTP {A1 3.675, A2 -64.154, A3 102.444, A4 32.455, A5 -52.928, A6 0.000, E1 766.66, E2 0, E3 0, E4 0, E5 0, E6 0} C_DIS
   SPTP {A1 3.702, A2 -63.247, A3 102.111, A4 31.530, A5 -55.143, A6 0.000, E1 769.75, E2 0, E3 0, E4 0, E5 0, E6 0} C_DIS
   SPTP {A1 3.748, A2 -62.309, A3 101.688, A4 30.809, A5 -57.343, A6 0.000, E1 772.67, E2 0, E3 0, E4 0, E5 0, E6 0} C_DIS
   SPTP {A1 3.847, A2 -61.696, A3 101.360, A4 30.621, A5 -58.781, A6 0.000, E1 775.05, E2 0, E3 0, E4 0, E5 0, E6 0} C_DIS
   SPTP {A1 3.975, A2 -61.187, A3 101.045, A4 30.669, A5 -59.964, A6 0.000, E1 777.21, E2 0, E3 0, E4 0, E5 0, E6 0} C_DIS
   SPTP {A1 4.120, A2 -60.668, A3 100.692, A4 30.820, A5 -61.134, A6 0.000, E1 779.3, E2 0, E3 0, E4 0, E5 0, E6 0} C_DIS
   SPTP {A1 4.278, A2 -60.142, A3 100.300, A4 31.064, A5 -62.290, A6 0.000, E1 781.32, E2 0, E3 0, E4 0, E5 0, E6 0} C_DIS
   SPTP {A1 4.449, A2 -59.609, A3 99.871, A4 31.390, A5 -63.425, A6 0.000, E1 783.28, E2 0, E3 0, E4 0, E5 0, E6 0} C_DIS
   SPTP {A1 4.630, A2 -59.070, A3 99.406, A4 31.792, A5 -64.540, A6 0.000, E1 785.19, E2 0, E3 0, E4 0, E5 0, E6 0} C_DIS
   SPTP {A1 4.821, A2 -58.527, A3 98.906, A4 32.260, A5 -65.632, A6 0.000, E1 787.05, E2 0, E3 0, E4 0, E5 0, E6 0} C_DIS
   SPTP {A1 5.019, A2 -57.979, A3 98.371, A4 32.789, A5 -66.699, A6 0.000, E1 788.87, E2 0, E3 0, E4 0, E5 0, E6 0} C_DIS
   SPTP {A1 5.291, A2 -57.806, A3 98.043, A4 33.761, A5 -67.029, A6 0.000, E1 790.33, E2 0, E3 0, E4 0, E5 0, E6 0} C_DIS
   SPTP {A1 5.569, A2 -57.636, A3 97.694, A4 34.786, A5 -67.337, A6 0.000, E1 791.73, E2 0, E3 0, E4 0, E5 0, E6 0} C_DIS
   SPTP {A1 5.851, A2 -57.463, A3 97.321, A4 35.853, A5 -67.634, A6 0.000, E1 793.1, E2 0, E3 0, E4 0, E5 0, E6 0} C_DIS
   SPTP {A1 6.135, A2 -57.288, A3 96.926, A4 36.955, A5 -67.921, A6 0.000, E1 794.44, E2 0, E3 0, E4 0, E5 0, E6 0} C_DIS
   SPTP {A1 6.421, A2 -57.109, A3 96.506, A4 38.089, A5 -68.197, A6 0.000, E1 795.75, E2 0, E3 0, E4 0, E5 0, E6 0} C_DIS
   SPTP {A1 6.706, A2 -56.928, A3 96.064, A4 39.250, A5 -68.462, A6 0.000, E1 797.02, E2 0, E3 0, E4 0, E5 0, E6 0} C_DIS
   SPTP {A1 6.989, A2 -56.745, A3 95.600, A4 40.432, A5 -68.717, A6 0.000, E1 798.28, E2 0, E3 0, E4 0, E5 0, E6 0} C_DIS
   SPTP {A1 7.270, A2 -56.559, A3 95.116, A4 41.632, A5 -68.962, A6 0.000, E1 799.51, E2 0, E3 0, E4 0, E5 0, E6 0} C_DIS
   SPTP {A1 7.547, A2 -56.372, A3 94.612, A4 42.845, A5 -69.196, A6 0.000, E1 800.72, E2 0, E3 0, E4 0, E5 0, E6 0} C_DIS
   SPTP {A1 7.819, A2 -56.185, A3 94.091, A4 44.067, A5 -69.419, A6 0.000, E1 801.92, E2 0, E3 0, E4 0, E5 0, E6 0} C_DIS
   SPTP {A1 8.085, A2 -55.996, A3 93.553, A4 45.297, A5 -69.631, A6 0.000, E1 803.11, E2 0, E3 0, E4 0, E5 0, E6 0} C_DIS
   SPTP {A1 8.349, A2 -55.845, A3 93.026, A4 46.565, A5 -69.770, A6 0.000, E1 804.23, E2 0, E3 0, E4 0, E5 0, E6 0} C_DIS
   SPTP {A1 8.615, A2 -55.779, A3 92.547, A4 47.924, A5 -69.755, A6 0.000, E1 805.19, E2 0, E3 0, E4 0, E5 0, E6 0} C_DIS
   SPTP {A1 8.873, A2 -55.713, A3 92.052, A4 49.286, A5 -69.736, A6 0.000, E1 806.15, E2 0, E3 0, E4 0, E5 0, E6 0} C_DIS
   SPTP {A1 9.123, A2 -55.644, A3 91.542, A4 50.650, A5 -69.712, A6 0.000, E1 807.09, E2 0, E3 0, E4 0, E5 0, E6 0} C_DIS
   SPTP {A1 9.364, A2 -55.575, A3 91.021, A4 52.011, A5 -69.683, A6 0.000, E1 808.02, E2 0, E3 0, E4 0, E5 0, E6 0} C_DIS
   SPTP {A1 9.596, A2 -55.505, A3 90.489, A4 53.367, A5 -69.649, A6 0.000, E1 808.95, E2 0, E3 0, E4 0, E5 0, E6 0} C_DIS
   SPTP {A1 9.819, A2 -55.437, A3 89.948, A4 54.717, A5 -69.609, A6 0.000, E1 809.87, E2 0, E3 0, E4 0, E5 0, E6 0} C_DIS
   SPTP {A1 10.031, A2 -55.371, A3 89.401, A4 56.059, A5 -69.563, A6 0.000, E1 810.79, E2 0, E3 0, E4 0, E5 0, E6 0} C_DIS
   SPTP {A1 10.233, A2 -55.308, A3 88.851, A4 57.388, A5 -69.509, A6 0.000, E1 811.71, E2 0, E3 0, E4 0, E5 0, E6 0} C_DIS
   SPTP {A1 10.424, A2 -55.248, A3 88.298, A4 58.706, A5 -69.447, A6 0.000, E1 812.62, E2 0, E3 0, E4 0, E5 0, E6 0} C_DIS
   SPTP {A1 10.603, A2 -55.194, A3 87.752, A4 59.998, A5 -69.378, A6 0.000, E1 813.54, E2 0, E3 0, E4 0, E5 0, E6 0} C_DIS
   SPTP {A1 10.759, A2 -55.147, A3 87.235, A4 61.218, A5 -69.319, A6 0.000, E1 814.44, E2 0, E3 0, E4 0, E5 0, E6 0} C_DIS
   SPTP {A1 10.896, A2 -55.108, A3 86.748, A4 62.369, A5 -69.267, A6 0.000, E1 815.33, E2 0, E3 0, E4 0, E5 0, E6 0} C_DIS
   SPTP {A1 11.005, A2 -55.078, A3 86.315, A4 63.402, A5 -69.238, A6 0.000, E1 816.19, E2 0, E3 0, E4 0, E5 0, E6 0} C_DIS
   SPTP {A1 11.106, A2 -55.056, A3 85.893, A4 64.418, A5 -69.196, A6 0.000, E1 817.06, E2 0, E3 0, E4 0, E5 0, E6 0} C_DIS
   SPTP {A1 11.198, A2 -55.044, A3 85.483, A4 65.415, A5 -69.139, A6 0.000, E1 817.94, E2 0, E3 0, E4 0, E5 0, E6 0} C_DIS
   SPTP {A1 11.282, A2 -55.045, A3 85.090, A4 66.391, A5 -69.064, A6 0.000, E1 818.84, E2 0, E3 0, E4 0, E5 0, E6 0} C_DIS
   SPTP {A1 11.357, A2 -55.058, A3 84.714, A4 67.347, A5 -68.970, A6 0.000, E1 819.76, E2 0, E3 0, E4 0, E5 0, E6 0} C_DIS
   SPTP {A1 11.424, A2 -55.084, A3 84.356, A4 68.282, A5 -68.857, A6 0.000, E1 820.69, E2 0, E3 0, E4 0, E5 0, E6 0} C_DIS
   SPTP {A1 11.483, A2 -55.124, A3 84.018, A4 69.197, A5 -68.723, A6 0.000, E1 821.63, E2 0, E3 0, E4 0, E5 0, E6 0} C_DIS
   SPTP {A1 11.534, A2 -55.177, A3 83.702, A4 70.091, A5 -68.569, A6 0.000, E1 822.59, E2 0, E3 0, E4 0, E5 0, E6 0} C_DIS
   SPTP {A1 11.576, A2 -55.246, A3 83.407, A4 70.965, A5 -68.392, A6 0.000, E1 823.56, E2 0, E3 0, E4 0, E5 0, E6 0} C_DIS
   SPTP {A1 11.610, A2 -55.330, A3 83.139, A4 71.816, A5 -68.191, A6 0.000, E1 824.55, E2 0, E3 0, E4 0, E5 0, E6 0} C_DIS
   SPTP {A1 11.637, A2 -55.431, A3 82.895, A4 72.646, A5 -67.966, A6 0.000, E1 825.56, E2 0, E3 0, E4 0, E5 0, E6 0} C_DIS
   SPTP {A1 11.655, A2 -55.549, A3 82.679, A4 73.454, A5 -67.713, A6 0.000, E1 826.59, E2 0, E3 0, E4 0, E5 0, E6 0} C_DIS
   SPTP {A1 11.665, A2 -55.685, A3 82.491, A4 74.240, A5 -67.433, A6 0.000, E1 827.63, E2 0, E3 0, E4 0, E5 0, E6 0} C_DIS
   SPTP {A1 11.667, A2 -55.837, A3 82.331, A4 75.005, A5 -67.125, A6 0.000, E1 828.69, E2 0, E3 0, E4 0, E5 0, E6 0} C_DIS
   SPTP {A1 11.661, A2 -56.007, A3 82.200, A4 75.748, A5 -66.790, A6 0.000, E1 829.76, E2 0, E3 0, E4 0, E5 0, E6 0} C_DIS
   SPTP {A1 11.647, A2 -56.195, A3 82.099, A4 76.470, A5 -66.425, A6 0.000, E1 830.85, E2 0, E3 0, E4 0, E5 0, E6 0} C_DIS
   SPTP {A1 11.622, A2 -56.421, A3 82.050, A4 77.187, A5 -66.019, A6 0.000, E1 831.82, E2 0, E3 0, E4 0, E5 0, E6 0} C_DIS
   SPTP {A1 11.584, A2 -56.695, A3 82.066, A4 77.907, A5 -65.565, A6 0.000, E1 832.62, E2 0, E3 0, E4 0, E5 0, E6 0} C_DIS
   SPTP {A1 11.540, A2 -56.980, A3 82.101, A4 78.614, A5 -65.090, A6 0.000, E1 833.42, E2 0, E3 0, E4 0, E5 0, E6 0} C_DIS
   SPTP {A1 11.487, A2 -57.279, A3 82.157, A4 79.306, A5 -64.589, A6 0.000, E1 834.23, E2 0, E3 0, E4 0, E5 0, E6 0} C_DIS
   SPTP {A1 11.428, A2 -57.591, A3 82.236, A4 79.983, A5 -64.062, A6 0.000, E1 835.04, E2 0, E3 0, E4 0, E5 0, E6 0} C_DIS
   SPTP {A1 11.360, A2 -57.915, A3 82.336, A4 80.647, A5 -63.510, A6 0.000, E1 835.86, E2 0, E3 0, E4 0, E5 0, E6 0} C_DIS
   SPTP {A1 11.285, A2 -58.253, A3 82.459, A4 81.295, A5 -62.929, A6 0.000, E1 836.69, E2 0, E3 0, E4 0, E5 0, E6 0} C_DIS
   SPTP {A1 11.202, A2 -58.604, A3 82.604, A4 81.928, A5 -62.320, A6 0.000, E1 837.52, E2 0, E3 0, E4 0, E5 0, E6 0} C_DIS
   SPTP {A1 11.110, A2 -58.967, A3 82.770, A4 82.547, A5 -61.684, A6 0.000, E1 838.36, E2 0, E3 0, E4 0, E5 0, E6 0} C_DIS
   SPTP {A1 11.011, A2 -59.342, A3 82.957, A4 83.152, A5 -61.019, A6 0.000, E1 839.2, E2 0, E3 0, E4 0, E5 0, E6 0} C_DIS
   SPTP {A1 10.903, A2 -59.728, A3 83.164, A4 83.744, A5 -60.326, A6 0.000, E1 840.04, E2 0, E3 0, E4 0, E5 0, E6 0} C_DIS
   SPTP {A1 10.786, A2 -60.125, A3 83.390, A4 84.322, A5 -59.605, A6 0.000, E1 840.89, E2 0, E3 0, E4 0, E5 0, E6 0} C_DIS
   SPTP {A1 10.666, A2 -60.569, A3 83.573, A4 85.186, A5 -58.780, A6 0.000, E1 841.4, E2 0, E3 0, E4 0, E5 0, E6 0} C_DIS
   SPTP {A1 10.539, A2 -61.045, A3 83.713, A4 86.290, A5 -57.881, A6 0.000, E1 841.63, E2 0, E3 0, E4 0, E5 0, E6 0} C_DIS
   SPTP {A1 10.400, A2 -61.521, A3 83.857, A4 87.409, A5 -56.971, A6 0.000, E1 841.84, E2 0, E3 0, E4 0, E5 0, E6 0} C_DIS
   SPTP {A1 10.249, A2 -62.001, A3 84.009, A4 88.539, A5 -56.043, A6 0.000, E1 842.01, E2 0, E3 0, E4 0, E5 0, E6 0} C_DIS
   SPTP {A1 10.087, A2 -62.482, A3 84.165, A4 89.684, A5 -55.102, A6 0.000, E1 842.16, E2 0, E3 0, E4 0, E5 0, E6 0} C_DIS
   SPTP {A1 9.913, A2 -62.963, A3 84.324, A4 90.848, A5 -54.150, A6 0.000, E1 842.28, E2 0, E3 0, E4 0, E5 0, E6 0} C_DIS
   SPTP {A1 9.726, A2 -63.443, A3 84.487, A4 92.032, A5 -53.186, A6 0.000, E1 842.37, E2 0, E3 0, E4 0, E5 0, E6 0} C_DIS
   SPTP {A1 9.528, A2 -63.923, A3 84.654, A4 93.238, A5 -52.210, A6 0.000, E1 842.42, E2 0, E3 0, E4 0, E5 0, E6 0} C_DIS
   SPTP {A1 9.318, A2 -64.402, A3 84.823, A4 94.469, A5 -51.224, A6 0.000, E1 842.43, E2 0, E3 0, E4 0, E5 0, E6 0} C_DIS
   SPTP {A1 9.095, A2 -64.879, A3 84.994, A4 95.728, A5 -50.229, A6 0.000, E1 842.4, E2 0, E3 0, E4 0, E5 0, E6 0} C_DIS
   SPTP {A1 8.860, A2 -65.353, A3 85.167, A4 97.018, A5 -49.227, A6 0.000, E1 842.33, E2 0, E3 0, E4 0, E5 0, E6 0} C_DIS
   SPTP {A1 8.614, A2 -65.824, A3 85.340, A4 98.343, A5 -48.218, A6 0.000, E1 842.21, E2 0, E3 0, E4 0, E5 0, E6 0} C_DIS
   SPTP {A1 8.355, A2 -66.291, A3 85.514, A4 99.705, A5 -47.203, A6 0.000, E1 842.05, E2 0, E3 0, E4 0, E5 0, E6 0} C_DIS
   SPTP {A1 8.084, A2 -66.753, A3 85.687, A4 101.109, A5 -46.186, A6 0.000, E1 841.83, E2 0, E3 0, E4 0, E5 0, E6 0} C_DIS
   SPTP {A1 7.802, A2 -67.208, A3 85.857, A4 102.560, A5 -45.170, A6 0.000, E1 841.56, E2 0, E3 0, E4 0, E5 0, E6 0} C_DIS
   SPTP {A1 7.494, A2 -67.667, A3 85.938, A4 104.451, A5 -44.089, A6 0.000, E1 841.02, E2 0, E3 0, E4 0, E5 0, E6 0} C_DIS
   SPTP {A1 7.170, A2 -68.118, A3 85.994, A4 106.505, A5 -43.012, A6 0.000, E1 840.35, E2 0, E3 0, E4 0, E5 0, E6 0} C_DIS
   SPTP {A1 6.831, A2 -68.557, A3 86.047, A4 108.640, A5 -41.955, A6 0.000, E1 839.6, E2 0, E3 0, E4 0, E5 0, E6 0} C_DIS
   SPTP {A1 6.477, A2 -68.985, A3 86.096, A4 110.862, A5 -40.921, A6 0.000, E1 838.74, E2 0, E3 0, E4 0, E5 0, E6 0} C_DIS
   SPTP {A1 6.110, A2 -69.400, A3 86.141, A4 113.174, A5 -39.917, A6 0.000, E1 837.8, E2 0, E3 0, E4 0, E5 0, E6 0} C_DIS
   SPTP {A1 5.729, A2 -69.801, A3 86.181, A4 115.581, A5 -38.946, A6 0.000, E1 836.75, E2 0, E3 0, E4 0, E5 0, E6 0} C_DIS
   SPTP {A1 5.338, A2 -70.188, A3 86.215, A4 118.085, A5 -38.018, A6 0.000, E1 835.6, E2 0, E3 0, E4 0, E5 0, E6 0} C_DIS
   SPTP {A1 4.936, A2 -70.558, A3 86.242, A4 120.685, A5 -37.140, A6 0.000, E1 834.36, E2 0, E3 0, E4 0, E5 0, E6 0} C_DIS
   SPTP {A1 4.525, A2 -70.912, A3 86.263, A4 123.382, A5 -36.317, A6 0.000, E1 833.02, E2 0, E3 0, E4 0, E5 0, E6 0} C_DIS
   SPTP {A1 4.107, A2 -71.250, A3 86.276, A4 126.170, A5 -35.555, A6 0.000, E1 831.6, E2 0, E3 0, E4 0, E5 0, E6 0} C_DIS
   SPTP {A1 3.682, A2 -71.570, A3 86.283, A4 129.042, A5 -34.861, A6 0.000, E1 830.09, E2 0, E3 0, E4 0, E5 0, E6 0} C_DIS
   SPTP {A1 3.252, A2 -71.874, A3 86.284, A4 131.995, A5 -34.232, A6 0.000, E1 828.51, E2 0, E3 0, E4 0, E5 0, E6 0} C_DIS
   SPTP {A1 2.819, A2 -72.161, A3 86.279, A4 135.008, A5 -33.683, A6 0.000, E1 826.89, E2 0, E3 0, E4 0, E5 0, E6 0} C_DIS
   SPTP {A1 2.387, A2 -72.452, A3 86.352, A4 137.889, A5 -33.083, A6 0.000, E1 825.45, E2 0, E3 0, E4 0, E5 0, E6 0} C_DIS
   SPTP {A1 1.951, A2 -72.828, A3 86.792, A4 140.072, A5 -31.947, A6 0.000, E1 824.89, E2 0, E3 0, E4 0, E5 0, E6 0} C_DIS
   SPTP {A1 1.518, A2 -73.192, A3 87.238, A4 142.330, A5 -30.835, A6 0.000, E1 824.26, E2 0, E3 0, E4 0, E5 0, E6 0} C_DIS
   SPTP {A1 1.090, A2 -73.544, A3 87.692, A4 144.663, A5 -29.749, A6 0.000, E1 823.56, E2 0, E3 0, E4 0, E5 0, E6 0} C_DIS
   SPTP {A1 0.672, A2 -73.885, A3 88.151, A4 147.056, A5 -28.699, A6 0.000, E1 822.82, E2 0, E3 0, E4 0, E5 0, E6 0} C_DIS
   SPTP {A1 0.266, A2 -74.213, A3 88.616, A4 149.495, A5 -27.687, A6 0.000, E1 822.04, E2 0, E3 0, E4 0, E5 0, E6 0} C_DIS
   SPTP {A1 -0.122, A2 -74.530, A3 89.089, A4 151.958, A5 -26.714, A6 0.000, E1 821.27, E2 0, E3 0, E4 0, E5 0, E6 0} C_DIS
   SPTP {A1 -0.489, A2 -74.837, A3 89.569, A4 154.418, A5 -25.781, A6 0.000, E1 820.52, E2 0, E3 0, E4 0, E5 0, E6 0} C_DIS
   SPTP {A1 -0.817, A2 -75.286, A3 90.751, A4 155.278, A5 -23.559, A6 0.000, E1 821.39, E2 0, E3 0, E4 0, E5 0, E6 0} C_DIS
   SPTP {A1 -1.116, A2 -75.705, A3 91.937, A4 155.975, A5 -21.302, A6 0.000, E1 822.44, E2 0, E3 0, E4 0, E5 0, E6 0} C_DIS
   SPTP {A1 -1.381, A2 -76.089, A3 93.106, A4 156.481, A5 -19.049, A6 0.000, E1 823.69, E2 0, E3 0, E4 0, E5 0, E6 0} C_DIS
   SPTP {A1 -1.601, A2 -76.437, A3 94.253, A4 156.610, A5 -16.815, A6 0.000, E1 825.34, E2 0, E3 0, E4 0, E5 0, E6 0} C_DIS
   SPTP {A1 -1.774, A2 -76.749, A3 95.382, A4 156.185, A5 -14.599, A6 0.000, E1 827.58, E2 0, E3 0, E4 0, E5 0, E6 0} C_DIS
   SPTP {A1 -1.893, A2 -77.058, A3 97.237, A4 150.120, A5 -10.711, A6 0.000, E1 835.41, E2 0, E3 0, E4 0, E5 0, E6 0} C_DIS
   SPTP {A1 -1.964, A2 -77.242, A3 98.996, A4 136.076, A5 -7.126, A6 0.000, E1 851.22, E2 0, E3 0, E4 0, E5 0, E6 0} C_DIS
   SPTP {A1 -1.984, A2 -77.295, A3 100.632, A4 101.397, A5 -4.820, A6 0.000, E1 887.68, E2 0, E3 0, E4 0, E5 0, E6 0} C_DIS
   SPTP {A1 -1.949, A2 -77.216, A3 102.140, A4 55.323, A5 -5.708, A6 0.000, E1 935.54, E2 0, E3 0, E4 0, E5 0, E6 0} C_DIS
   SPTP {A1 -1.868, A2 -76.864, A3 103.815, A4 29.166, A5 -9.944, A6 0.000, E1 963.5, E2 0, E3 0, E4 0, E5 0, E6 0} C_DIS
   SPTP {A1 -1.750, A2 -76.122, A3 105.466, A4 18.831, A5 -16.042, A6 0.000, E1 975.65, E2 0, E3 0, E4 0, E5 0, E6 0} C_DIS
   SPTP {A1 -1.596, A2 -75.081, A3 106.761, A4 14.729, A5 -22.370, A6 0.000, E1 981.56, E2 0, E3 0, E4 0, E5 0, E6 0} C_DIS
   SPTP {A1 -1.420, A2 -73.679, A3 107.713, A4 12.621, A5 -29.006, A6 0.000, E1 985.51, E2 0, E3 0, E4 0, E5 0, E6 0} C_DIS
   SPTP {A1 -1.228, A2 -71.398, A3 108.266, A4 10.959, A5 -37.420, A6 0.000, E1 989.3, E2 0, E3 0, E4 0, E5 0, E6 0} C_DIS
   SPTP {A1 -1.030, A2 -68.707, A3 108.117, A4 10.162, A5 -45.592, A6 0.000, E1 992.22, E2 0, E3 0, E4 0, E5 0, E6 0} C_DIS
   SPTP {A1 -0.838, A2 -65.683, A3 107.265, A4 9.810, A5 -53.419, A6 0.000, E1 994.72, E2 0, E3 0, E4 0, E5 0, E6 0} C_DIS
   SPTP {A1 -0.649, A2 -62.454, A3 105.747, A4 9.736, A5 -60.713, A6 0.000, E1 997.03, E2 0, E3 0, E4 0, E5 0, E6 0} C_DIS
   SPTP {A1 -0.240, A2 -59.801, A3 104.073, A4 10.496, A5 -66.108, A6 0.000, E1 999.44, E2 0, E3 0, E4 0, E5 0, E6 0} C_DIS
   SPTP {A1 0.183, A2 -57.088, A3 101.995, A4 11.405, A5 -71.139, A6 0.000, E1 1001.8, E2 0, E3 0, E4 0, E5 0, E6 0} C_DIS
   SPTP {A1 0.621, A2 -54.343, A3 99.532, A4 12.465, A5 -75.792, A6 0.000, E1 1004.11, E2 0, E3 0, E4 0, E5 0, E6 0} C_DIS
   SPTP {A1 1.069, A2 -51.589, A3 96.701, A4 13.660, A5 -80.060, A6 0.000, E1 1006.4, E2 0, E3 0, E4 0, E5 0, E6 0} C_DIS
   SPTP {A1 1.523, A2 -48.843, A3 93.524, A4 14.975, A5 -83.940, A6 0.000, E1 1008.66, E2 0, E3 0, E4 0, E5 0, E6 0} C_DIS
   SPTP {A1 1.981, A2 -46.107, A3 90.005, A4 16.417, A5 -87.438, A6 0.000, E1 1010.89, E2 0, E3 0, E4 0, E5 0, E6 0} C_DIS
   SPTP {A1 2.446, A2 -43.377, A3 86.146, A4 17.993, A5 -90.566, A6 0.000, E1 1013.07, E2 0, E3 0, E4 0, E5 0, E6 0} C_DIS
   SPTP {A1 2.910, A2 -40.644, A3 81.941, A4 19.684, A5 -93.330, A6 0.000, E1 1015.18, E2 0, E3 0, E4 0, E5 0, E6 0} C_DIS
   SPTP {A1 3.372, A2 -37.887, A3 77.367, A4 21.485, A5 -95.741, A6 0.000, E1 1017.2, E2 0, E3 0, E4 0, E5 0, E6 0} C_DIS
   SPTP {A1 3.827, A2 -35.072, A3 72.380, A4 23.379, A5 -97.802, A6 0.000, E1 1019.09, E2 0, E3 0, E4 0, E5 0, E6 0} C_DIS
   SPTP {A1 4.388, A2 -34.778, A3 71.371, A4 25.533, A5 -97.859, A6 0.000, E1 1020.43, E2 0, E3 0, E4 0, E5 0, E6 0} C_DIS
   SPTP {A1 4.950, A2 -34.657, A3 70.589, A4 27.772, A5 -97.748, A6 0.000, E1 1021.58, E2 0, E3 0, E4 0, E5 0, E6 0} C_DIS
   SPTP {A1 5.502, A2 -34.512, A3 69.715, A4 30.064, A5 -97.608, A6 0.000, E1 1022.59, E2 0, E3 0, E4 0, E5 0, E6 0} C_DIS
   SPTP {A1 6.026, A2 -34.589, A3 69.190, A4 32.324, A5 -97.302, A6 0.000, E1 1023.37, E2 0, E3 0, E4 0, E5 0, E6 0} C_DIS
   SPTP {A1 6.504, A2 -35.243, A3 69.653, A4 34.453, A5 -96.620, A6 0.000, E1 1023.76, E2 0, E3 0, E4 0, E5 0, E6 0} C_DIS
   SPTP {A1 6.974, A2 -35.850, A3 69.990, A4 36.617, A5 -95.927, A6 0.000, E1 1024.04, E2 0, E3 0, E4 0, E5 0, E6 0} C_DIS
   SPTP {A1 7.206, A2 -36.138, A3 70.118, A4 37.711, A5 -95.577, A6 0.000, E1 1024.14, E2 0, E3 0, E4 0, E5 0, E6 0} C_DIS
   SPTP {A1 7.434, A2 -36.418, A3 70.220, A4 38.809, A5 -95.225, A6 0.000, E1 1024.21, E2 0, E3 0, E4 0, E5 0, E6 0} C_DIS
   SPTP {A1 7.435, A2 -36.403, A3 70.202, A4 38.822, A5 -95.236, A6 0.000, E1 1024.19, E2 0, E3 0, E4 0, E5 0, E6 0} C_DIS
   SPTP {A1 7.883, A2 -36.938, A3 70.338, A4 41.019, A5 -94.529, A6 0.000, E1 1024.29, E2 0, E3 0, E4 0, E5 0, E6 0} C_DIS
   SPTP {A1 8.286, A2 -37.718, A3 70.895, A4 43.080, A5 -93.650, A6 0.000, E1 1024.14, E2 0, E3 0, E4 0, E5 0, E6 0} C_DIS
   SPTP {A1 8.649, A2 -38.737, A3 71.850, A4 45.018, A5 -92.589, A6 0.000, E1 1023.72, E2 0, E3 0, E4 0, E5 0, E6 0} C_DIS
   SPTP {A1 9.005, A2 -39.719, A3 72.693, A4 46.976, A5 -91.508, A6 0.000, E1 1023.22, E2 0, E3 0, E4 0, E5 0, E6 0} C_DIS
   SPTP {A1 9.352, A2 -40.671, A3 73.436, A4 48.956, A5 -90.413, A6 0.000, E1 1022.65, E2 0, E3 0, E4 0, E5 0, E6 0} C_DIS
   SPTP {A1 9.690, A2 -41.597, A3 74.095, A4 50.945, A5 -89.304, A6 0.000, E1 1022.03, E2 0, E3 0, E4 0, E5 0, E6 0} C_DIS
   SPTP {A1 10.015, A2 -42.506, A3 74.683, A4 52.943, A5 -88.178, A6 0.000, E1 1021.36, E2 0, E3 0, E4 0, E5 0, E6 0} C_DIS
   SPTP {A1 10.326, A2 -43.402, A3 75.212, A4 54.944, A5 -87.036, A6 0.000, E1 1020.65, E2 0, E3 0, E4 0, E5 0, E6 0} C_DIS
   SPTP {A1 10.622, A2 -44.288, A3 75.689, A4 56.946, A5 -85.877, A6 0.000, E1 1019.9, E2 0, E3 0, E4 0, E5 0, E6 0} C_DIS
   SPTP {A1 10.877, A2 -45.277, A3 76.330, A4 58.849, A5 -84.635, A6 0.000, E1 1018.93, E2 0, E3 0, E4 0, E5 0, E6 0} C_DIS
   SPTP {A1 11.108, A2 -46.304, A3 77.002, A4 60.722, A5 -83.343, A6 0.000, E1 1017.84, E2 0, E3 0, E4 0, E5 0, E6 0} C_DIS
   SPTP {A1 11.324, A2 -47.299, A3 77.585, A4 62.632, A5 -82.058, A6 0.000, E1 1016.66, E2 0, E3 0, E4 0, E5 0, E6 0} C_DIS
   SPTP {A1 11.522, A2 -48.289, A3 78.119, A4 64.555, A5 -80.756, A6 0.000, E1 1015.43, E2 0, E3 0, E4 0, E5 0, E6 0} C_DIS
   SPTP {A1 11.702, A2 -49.259, A3 78.589, A4 66.508, A5 -79.456, A6 0.000, E1 1014.13, E2 0, E3 0, E4 0, E5 0, E6 0} C_DIS
   SPTP {A1 11.860, A2 -50.222, A3 79.013, A4 68.480, A5 -78.146, A6 0.000, E1 1012.77, E2 0, E3 0, E4 0, E5 0, E6 0} C_DIS
   SPTP {A1 11.997, A2 -51.170, A3 79.382, A4 70.482, A5 -76.837, A6 0.000, E1 1011.34, E2 0, E3 0, E4 0, E5 0, E6 0} C_DIS
   SPTP {A1 12.112, A2 -52.099, A3 79.694, A4 72.521, A5 -75.540, A6 0.000, E1 1009.83, E2 0, E3 0, E4 0, E5 0, E6 0} C_DIS
   SPTP {A1 12.202, A2 -53.016, A3 79.960, A4 74.593, A5 -74.246, A6 0.000, E1 1008.24, E2 0, E3 0, E4 0, E5 0, E6 0} C_DIS
   SPTP {A1 12.269, A2 -53.905, A3 80.159, A4 76.717, A5 -72.983, A6 0.000, E1 1006.56, E2 0, E3 0, E4 0, E5 0, E6 0} C_DIS
   SPTP {A1 12.308, A2 -54.781, A3 80.314, A4 78.881, A5 -71.732, A6 0.000, E1 1004.8, E2 0, E3 0, E4 0, E5 0, E6 0} C_DIS
   SPTP {A1 12.324, A2 -55.618, A3 80.392, A4 81.112, A5 -70.534, A6 0.000, E1 1002.93, E2 0, E3 0, E4 0, E5 0, E6 0} C_DIS
   SPTP {A1 12.312, A2 -56.438, A3 80.425, A4 83.391, A5 -69.362, A6 0.000, E1 1000.97, E2 0, E3 0, E4 0, E5 0, E6 0} C_DIS
   SPTP {A1 12.273, A2 -57.203, A3 80.384, A4 85.696, A5 -68.271, A6 0.000, E1 998.99, E2 0, E3 0, E4 0, E5 0, E6 0} C_DIS
   SPTP {A1 12.204, A2 -57.886, A3 80.335, A4 87.782, A5 -67.261, A6 0.000, E1 997.48, E2 0, E3 0, E4 0, E5 0, E6 0} C_DIS
   SPTP {A1 12.111, A2 -58.545, A3 80.255, A4 89.894, A5 -66.286, A6 0.000, E1 995.95, E2 0, E3 0, E4 0, E5 0, E6 0} C_DIS
   SPTP {A1 11.993, A2 -59.187, A3 80.146, A4 92.051, A5 -65.345, A6 0.000, E1 994.34, E2 0, E3 0, E4 0, E5 0, E6 0} C_DIS
   SPTP {A1 11.852, A2 -59.805, A3 80.000, A4 94.261, A5 -64.446, A6 0.000, E1 992.65, E2 0, E3 0, E4 0, E5 0, E6 0} C_DIS
   SPTP {A1 11.688, A2 -60.395, A3 79.812, A4 96.527, A5 -63.603, A6 0.000, E1 990.89, E2 0, E3 0, E4 0, E5 0, E6 0} C_DIS
   SPTP {A1 11.500, A2 -60.956, A3 79.581, A4 98.851, A5 -62.822, A6 0.000, E1 989.04, E2 0, E3 0, E4 0, E5 0, E6 0} C_DIS
   SPTP {A1 11.292, A2 -61.479, A3 79.295, A4 101.234, A5 -62.122, A6 0.000, E1 987.11, E2 0, E3 0, E4 0, E5 0, E6 0} C_DIS
   SPTP {A1 11.064, A2 -61.962, A3 78.979, A4 103.621, A5 -61.494, A6 0.000, E1 985.22, E2 0, E3 0, E4 0, E5 0, E6 0} C_DIS
   SPTP {A1 10.818, A2 -62.454, A3 78.917, A4 105.472, A5 -60.697, A6 0.000, E1 984.38, E2 0, E3 0, E4 0, E5 0, E6 0} C_DIS
   SPTP {A1 10.555, A2 -62.935, A3 78.846, A4 107.361, A5 -59.922, A6 0.000, E1 983.49, E2 0, E3 0, E4 0, E5 0, E6 0} C_DIS
   SPTP {A1 10.277, A2 -63.399, A3 78.761, A4 109.293, A5 -59.181, A6 0.000, E1 982.56, E2 0, E3 0, E4 0, E5 0, E6 0} C_DIS
   SPTP {A1 9.985, A2 -63.839, A3 78.653, A4 111.269, A5 -58.490, A6 0.000, E1 981.57, E2 0, E3 0, E4 0, E5 0, E6 0} C_DIS
   SPTP {A1 9.683, A2 -64.252, A3 78.514, A4 113.287, A5 -57.863, A6 0.000, E1 980.55, E2 0, E3 0, E4 0, E5 0, E6 0} C_DIS
   SPTP {A1 9.372, A2 -64.634, A3 78.342, A4 115.346, A5 -57.311, A6 0.000, E1 979.49, E2 0, E3 0, E4 0, E5 0, E6 0} C_DIS
   SPTP {A1 9.057, A2 -65.076, A3 78.457, A4 116.954, A5 -56.499, A6 0.000, E1 979.22, E2 0, E3 0, E4 0, E5 0, E6 0} C_DIS
   SPTP {A1 8.737, A2 -65.589, A3 78.864, A4 118.134, A5 -55.395, A6 0.000, E1 979.67, E2 0, E3 0, E4 0, E5 0, E6 0} C_DIS
   SPTP {A1 8.416, A2 -66.086, A3 79.267, A4 119.326, A5 -54.308, A6 0.000, E1 980.12, E2 0, E3 0, E4 0, E5 0, E6 0} C_DIS
   SPTP {A1 8.095, A2 -66.566, A3 79.662, A4 120.527, A5 -53.246, A6 0.000, E1 980.56, E2 0, E3 0, E4 0, E5 0, E6 0} C_DIS
   SPTP {A1 7.776, A2 -67.028, A3 80.050, A4 121.735, A5 -52.212, A6 0.000, E1 981.01, E2 0, E3 0, E4 0, E5 0, E6 0} C_DIS
   SPTP {A1 7.463, A2 -67.511, A3 80.568, A4 122.712, A5 -51.053, A6 0.000, E1 981.8, E2 0, E3 0, E4 0, E5 0, E6 0} C_DIS
   SPTP {A1 7.163, A2 -68.158, A3 81.730, A4 122.567, A5 -49.160, A6 0.000, E1 984.17, E2 0, E3 0, E4 0, E5 0, E6 0} C_DIS
   SPTP {A1 6.870, A2 -68.774, A3 82.877, A4 122.308, A5 -47.280, A6 0.000, E1 986.63, E2 0, E3 0, E4 0, E5 0, E6 0} C_DIS
   SPTP {A1 6.588, A2 -69.355, A3 84.004, A4 121.921, A5 -45.424, A6 0.000, E1 989.22, E2 0, E3 0, E4 0, E5 0, E6 0} C_DIS
   SPTP {A1 6.318, A2 -69.901, A3 85.111, A4 121.392, A5 -43.596, A6 0.000, E1 991.93, E2 0, E3 0, E4 0, E5 0, E6 0} C_DIS
   SPTP {A1 6.063, A2 -70.443, A3 86.359, A4 120.290, A5 -41.620, A6 0.000, E1 995.29, E2 0, E3 0, E4 0, E5 0, E6 0} C_DIS
   SPTP {A1 5.827, A2 -71.035, A3 88.153, A4 117.295, A5 -39.061, A6 0.000, E1 1000.84, E2 0, E3 0, E4 0, E5 0, E6 0} C_DIS
   SPTP {A1 5.604, A2 -71.529, A3 89.861, A4 113.731, A5 -36.691, A6 0.000, E1 1006.91, E2 0, E3 0, E4 0, E5 0, E6 0} C_DIS
   SPTP {A1 5.393, A2 -71.926, A3 91.481, A4 109.544, A5 -34.550, A6 0.000, E1 1013.57, E2 0, E3 0, E4 0, E5 0, E6 0} C_DIS
   SPTP {A1 5.194, A2 -72.224, A3 93.010, A4 104.702, A5 -32.690, A6 0.000, E1 1020.85, E2 0, E3 0, E4 0, E5 0, E6 0} C_DIS
   SPTP {A1 5.010, A2 -72.423, A3 94.442, A4 99.215, A5 -31.175, A6 0.000, E1 1028.75, E2 0, E3 0, E4 0, E5 0, E6 0} C_DIS
   SPTP {A1 4.839, A2 -72.498, A3 95.886, A4 92.425, A5 -30.091, A6 0.000, E1 1037.89, E2 0, E3 0, E4 0, E5 0, E6 0} C_DIS
   SPTP {A1 4.676, A2 -72.427, A3 97.292, A4 84.589, A5 -29.611, A6 0.000, E1 1048.03, E2 0, E3 0, E4 0, E5 0, E6 0} C_DIS
   SPTP {A1 4.520, A2 -72.224, A3 98.549, A4 76.660, A5 -29.771, A6 0.000, E1 1058.23, E2 0, E3 0, E4 0, E5 0, E6 0} C_DIS
   SPTP {A1 4.371, A2 -71.891, A3 99.655, A4 69.005, A5 -30.553, A6 0.000, E1 1068.15, E2 0, E3 0, E4 0, E5 0, E6 0} C_DIS
   SPTP {A1 4.232, A2 -71.428, A3 100.603, A4 61.939, A5 -31.909, A6 0.000, E1 1077.47, E2 0, E3 0, E4 0, E5 0, E6 0} C_DIS
   SPTP {A1 4.106, A2 -70.840, A3 101.387, A4 55.664, A5 -33.762, A6 0.000, E1 1085.99, E2 0, E3 0, E4 0, E5 0, E6 0} C_DIS
   SPTP {A1 3.993, A2 -70.131, A3 102.006, A4 50.233, A5 -36.010, A6 0.000, E1 1093.69, E2 0, E3 0, E4 0, E5 0, E6 0} C_DIS
   SPTP {A1 3.894, A2 -69.309, A3 102.459, A4 45.621, A5 -38.563, A6 0.000, E1 1100.57, E2 0, E3 0, E4 0, E5 0, E6 0} C_DIS
   SPTP {A1 3.812, A2 -68.380, A3 102.741, A4 41.769, A5 -41.344, A6 0.000, E1 1106.71, E2 0, E3 0, E4 0, E5 0, E6 0} C_DIS
   SPTP {A1 3.749, A2 -67.419, A3 102.862, A4 38.731, A5 -44.112, A6 0.000, E1 1112.01, E2 0, E3 0, E4 0, E5 0, E6 0} C_DIS
   SPTP {A1 3.698, A2 -66.680, A3 102.904, A4 36.719, A5 -46.235, A6 0.000, E1 1116.04, E2 0, E3 0, E4 0, E5 0, E6 0} C_DIS
   SPTP {A1 3.667, A2 -65.894, A3 102.853, A4 35.024, A5 -48.407, A6 0.000, E1 1119.79, E2 0, E3 0, E4 0, E5 0, E6 0} C_DIS
   SPTP {A1 3.657, A2 -65.065, A3 102.706, A4 33.615, A5 -50.609, A6 0.000, E1 1123.28, E2 0, E3 0, E4 0, E5 0, E6 0} C_DIS
   SPTP {A1 3.666, A2 -64.196, A3 102.468, A4 32.459, A5 -52.824, A6 0.000, E1 1126.56, E2 0, E3 0, E4 0, E5 0, E6 0} C_DIS
   SPTP {A1 3.694, A2 -63.291, A3 102.138, A4 31.531, A5 -55.038, A6 0.000, E1 1129.64, E2 0, E3 0, E4 0, E5 0, E6 0} C_DIS
   SPTP {A1 3.740, A2 -62.354, A3 101.719, A4 30.807, A5 -57.239, A6 0.000, E1 1132.56, E2 0, E3 0, E4 0, E5 0, E6 0} C_DIS
   SPTP {A1 3.837, A2 -61.720, A3 101.382, A4 30.596, A5 -58.723, A6 0.000, E1 1134.96, E2 0, E3 0, E4 0, E5 0, E6 0} C_DIS
   SPTP {A1 3.964, A2 -61.211, A3 101.070, A4 30.642, A5 -59.907, A6 0.000, E1 1137.13, E2 0, E3 0, E4 0, E5 0, E6 0} C_DIS
   SPTP {A1 4.109, A2 -60.693, A3 100.717, A4 30.792, A5 -61.078, A6 0.000, E1 1139.21, E2 0, E3 0, E4 0, E5 0, E6 0} C_DIS
   SPTP {A1 4.267, A2 -60.167, A3 100.327, A4 31.036, A5 -62.234, A6 0.000, E1 1141.23, E2 0, E3 0, E4 0, E5 0, E6 0} C_DIS
   SPTP {A1 4.438, A2 -59.635, A3 99.899, A4 31.361, A5 -63.370, A6 0.000, E1 1143.19, E2 0, E3 0, E4 0, E5 0, E6 0} C_DIS
   SPTP {A1 4.619, A2 -59.096, A3 99.436, A4 31.761, A5 -64.486, A6 0.000, E1 1145.1, E2 0, E3 0, E4 0, E5 0, E6 0} C_DIS
   SPTP {A1 4.809, A2 -58.553, A3 98.937, A4 32.227, A5 -65.578, A6 0.000, E1 1146.96, E2 0, E3 0, E4 0, E5 0, E6 0} C_DIS
   SPTP {A1 5.008, A2 -58.006, A3 98.404, A4 32.756, A5 -66.646, A6 0.000, E1 1148.78, E2 0, E3 0, E4 0, E5 0, E6 0} C_DIS
   SPTP {A1 5.275, A2 -57.812, A3 98.064, A4 33.704, A5 -67.017, A6 0.000, E1 1150.25, E2 0, E3 0, E4 0, E5 0, E6 0} C_DIS
   SPTP {A1 5.554, A2 -57.641, A3 97.716, A4 34.728, A5 -67.326, A6 0.000, E1 1151.66, E2 0, E3 0, E4 0, E5 0, E6 0} C_DIS
   SPTP {A1 5.836, A2 -57.468, A3 97.344, A4 35.794, A5 -67.624, A6 0.000, E1 1153.03, E2 0, E3 0, E4 0, E5 0, E6 0} C_DIS
   SPTP {A1 6.120, A2 -57.293, A3 96.950, A4 36.893, A5 -67.912, A6 0.000, E1 1154.37, E2 0, E3 0, E4 0, E5 0, E6 0} C_DIS
   SPTP {A1 6.405, A2 -57.115, A3 96.531, A4 38.026, A5 -68.188, A6 0.000, E1 1155.67, E2 0, E3 0, E4 0, E5 0, E6 0} C_DIS
   SPTP {A1 6.690, A2 -56.933, A3 96.090, A4 39.185, A5 -68.455, A6 0.000, E1 1156.95, E2 0, E3 0, E4 0, E5 0, E6 0} C_DIS
   SPTP {A1 6.974, A2 -56.750, A3 95.627, A4 40.366, A5 -68.711, A6 0.000, E1 1158.2, E2 0, E3 0, E4 0, E5 0, E6 0} C_DIS
   SPTP {A1 7.255, A2 -56.564, A3 95.144, A4 41.565, A5 -68.956, A6 0.000, E1 1159.43, E2 0, E3 0, E4 0, E5 0, E6 0} C_DIS
   SPTP {A1 7.532, A2 -56.377, A3 94.642, A4 42.777, A5 -69.191, A6 0.000, E1 1160.65, E2 0, E3 0, E4 0, E5 0, E6 0} C_DIS
   SPTP {A1 7.804, A2 -56.189, A3 94.121, A4 43.999, A5 -69.415, A6 0.000, E1 1161.84, E2 0, E3 0, E4 0, E5 0, E6 0} C_DIS
   SPTP {A1 8.070, A2 -56.001, A3 93.584, A4 45.227, A5 -69.627, A6 0.000, E1 1163.03, E2 0, E3 0, E4 0, E5 0, E6 0} C_DIS
   SPTP {A1 8.333, A2 -55.841, A3 93.053, A4 46.486, A5 -69.781, A6 0.000, E1 1164.16, E2 0, E3 0, E4 0, E5 0, E6 0} C_DIS
   SPTP {A1 8.599, A2 -55.776, A3 92.575, A4 47.844, A5 -69.767, A6 0.000, E1 1165.13, E2 0, E3 0, E4 0, E5 0, E6 0} C_DIS
   SPTP {A1 8.858, A2 -55.709, A3 92.082, A4 49.205, A5 -69.747, A6 0.000, E1 1166.08, E2 0, E3 0, E4 0, E5 0, E6 0} C_DIS
   SPTP {A1 9.108, A2 -55.641, A3 91.574, A4 50.567, A5 -69.724, A6 0.000, E1 1167.02, E2 0, E3 0, E4 0, E5 0, E6 0} C_DIS
   SPTP {A1 9.350, A2 -55.572, A3 91.053, A4 51.926, A5 -69.696, A6 0.000, E1 1167.96, E2 0, E3 0, E4 0, E5 0, E6 0} C_DIS
   SPTP {A1 9.582, A2 -55.503, A3 90.522, A4 53.282, A5 -69.662, A6 0.000, E1 1168.88, E2 0, E3 0, E4 0, E5 0, E6 0} C_DIS
   SPTP {A1 9.805, A2 -55.434, A3 89.983, A4 54.631, A5 -69.623, A6 0.000, E1 1169.8, E2 0, E3 0, E4 0, E5 0, E6 0} C_DIS
   SPTP {A1 10.018, A2 -55.368, A3 89.436, A4 55.972, A5 -69.577, A6 0.000, E1 1170.72, E2 0, E3 0, E4 0, E5 0, E6 0} C_DIS
   SPTP {A1 10.220, A2 -55.304, A3 88.887, A4 57.301, A5 -69.523, A6 0.000, E1 1171.64, E2 0, E3 0, E4 0, E5 0, E6 0} C_DIS
   SPTP {A1 10.412, A2 -55.245, A3 88.335, A4 58.618, A5 -69.461, A6 0.000, E1 1172.56, E2 0, E3 0, E4 0, E5 0, E6 0} C_DIS
   SPTP {A1 10.592, A2 -55.190, A3 87.786, A4 59.915, A5 -69.393, A6 0.000, E1 1173.48, E2 0, E3 0, E4 0, E5 0, E6 0} C_DIS
   SPTP {A1 10.749, A2 -55.143, A3 87.269, A4 61.135, A5 -69.333, A6 0.000, E1 1174.37, E2 0, E3 0, E4 0, E5 0, E6 0} C_DIS
   SPTP {A1 10.889, A2 -55.103, A3 86.777, A4 62.297, A5 -69.278, A6 0.000, E1 1175.26, E2 0, E3 0, E4 0, E5 0, E6 0} C_DIS
   SPTP {A1 10.998, A2 -55.073, A3 86.344, A4 63.330, A5 -69.250, A6 0.000, E1 1176.12, E2 0, E3 0, E4 0, E5 0, E6 0} C_DIS
   SPTP {A1 11.099, A2 -55.051, A3 85.922, A4 64.346, A5 -69.209, A6 0.000, E1 1176.99, E2 0, E3 0, E4 0, E5 0, E6 0} C_DIS
   SPTP {A1 11.192, A2 -55.038, A3 85.512, A4 65.343, A5 -69.153, A6 0.000, E1 1177.88, E2 0, E3 0, E4 0, E5 0, E6 0} C_DIS
   SPTP {A1 11.277, A2 -55.038, A3 85.118, A4 66.320, A5 -69.079, A6 0.000, E1 1178.78, E2 0, E3 0, E4 0, E5 0, E6 0} C_DIS
   SPTP {A1 11.353, A2 -55.050, A3 84.740, A4 67.277, A5 -68.987, A6 0.000, E1 1179.69, E2 0, E3 0, E4 0, E5 0, E6 0} C_DIS
   SPTP {A1 11.420, A2 -55.075, A3 84.381, A4 68.213, A5 -68.875, A6 0.000, E1 1180.61, E2 0, E3 0, E4 0, E5 0, E6 0} C_DIS
   SPTP {A1 11.480, A2 -55.114, A3 84.042, A4 69.128, A5 -68.743, A6 0.000, E1 1181.56, E2 0, E3 0, E4 0, E5 0, E6 0} C_DIS
   SPTP {A1 11.531, A2 -55.167, A3 83.725, A4 70.023, A5 -68.590, A6 0.000, E1 1182.51, E2 0, E3 0, E4 0, E5 0, E6 0} C_DIS
   SPTP {A1 11.574, A2 -55.234, A3 83.429, A4 70.897, A5 -68.415, A6 0.000, E1 1183.49, E2 0, E3 0, E4 0, E5 0, E6 0} C_DIS
   SPTP {A1 11.609, A2 -55.317, A3 83.159, A4 71.749, A5 -68.216, A6 0.000, E1 1184.48, E2 0, E3 0, E4 0, E5 0, E6 0} C_DIS
   SPTP {A1 11.636, A2 -55.416, A3 82.913, A4 72.581, A5 -67.993, A6 0.000, E1 1185.48, E2 0, E3 0, E4 0, E5 0, E6 0} C_DIS
   SPTP {A1 11.655, A2 -55.532, A3 82.695, A4 73.391, A5 -67.744, A6 0.000, E1 1186.5, E2 0, E3 0, E4 0, E5 0, E6 0} C_DIS
   SPTP {A1 11.665, A2 -55.666, A3 82.504, A4 74.178, A5 -67.466, A6 0.000, E1 1187.54, E2 0, E3 0, E4 0, E5 0, E6 0} C_DIS
   SPTP {A1 11.668, A2 -55.817, A3 82.342, A4 74.944, A5 -67.161, A6 0.000, E1 1188.6, E2 0, E3 0, E4 0, E5 0, E6 0} C_DIS
   SPTP {A1 11.663, A2 -55.986, A3 82.209, A4 75.688, A5 -66.828, A6 0.000, E1 1189.67, E2 0, E3 0, E4 0, E5 0, E6 0} C_DIS
   SPTP {A1 11.650, A2 -56.172, A3 82.105, A4 76.411, A5 -66.466, A6 0.000, E1 1190.76, E2 0, E3 0, E4 0, E5 0, E6 0} C_DIS
   SPTP {A1 11.626, A2 -56.392, A3 82.049, A4 77.126, A5 -66.066, A6 0.000, E1 1191.76, E2 0, E3 0, E4 0, E5 0, E6 0} C_DIS
   SPTP {A1 11.589, A2 -56.664, A3 82.062, A4 77.847, A5 -65.614, A6 0.000, E1 1192.55, E2 0, E3 0, E4 0, E5 0, E6 0} C_DIS
   SPTP {A1 11.545, A2 -56.949, A3 82.095, A4 78.554, A5 -65.141, A6 0.000, E1 1193.35, E2 0, E3 0, E4 0, E5 0, E6 0} C_DIS
   SPTP {A1 11.493, A2 -57.246, A3 82.149, A4 79.248, A5 -64.644, A6 0.000, E1 1194.16, E2 0, E3 0, E4 0, E5 0, E6 0} C_DIS
   SPTP {A1 11.435, A2 -57.556, A3 82.226, A4 79.927, A5 -64.120, A6 0.000, E1 1194.97, E2 0, E3 0, E4 0, E5 0, E6 0} C_DIS
   SPTP {A1 11.368, A2 -57.878, A3 82.323, A4 80.592, A5 -63.572, A6 0.000, E1 1195.79, E2 0, E3 0, E4 0, E5 0, E6 0} C_DIS
   SPTP {A1 11.294, A2 -58.214, A3 82.443, A4 81.241, A5 -62.996, A6 0.000, E1 1196.61, E2 0, E3 0, E4 0, E5 0, E6 0} C_DIS
   SPTP {A1 11.212, A2 -58.563, A3 82.585, A4 81.876, A5 -62.390, A6 0.000, E1 1197.45, E2 0, E3 0, E4 0, E5 0, E6 0} C_DIS
   SPTP {A1 11.121, A2 -58.925, A3 82.749, A4 82.496, A5 -61.757, A6 0.000, E1 1198.28, E2 0, E3 0, E4 0, E5 0, E6 0} C_DIS
   SPTP {A1 11.022, A2 -59.298, A3 82.934, A4 83.102, A5 -61.096, A6 0.000, E1 1199.12, E2 0, E3 0, E4 0, E5 0, E6 0} C_DIS
   SPTP {A1 10.916, A2 -59.683, A3 83.138, A4 83.695, A5 -60.407, A6 0.000, E1 1199.97, E2 0, E3 0, E4 0, E5 0, E6 0} C_DIS
   SPTP {A1 10.800, A2 -60.078, A3 83.363, A4 84.274, A5 -59.689, A6 0.000, E1 1200.82, E2 0, E3 0, E4 0, E5 0, E6 0} C_DIS
   SPTP {A1 10.680, A2 -60.515, A3 83.554, A4 85.089, A5 -58.880, A6 0.000, E1 1201.38, E2 0, E3 0, E4 0, E5 0, E6 0} C_DIS
   SPTP {A1 10.554, A2 -60.990, A3 83.694, A4 86.191, A5 -57.983, A6 0.000, E1 1201.62, E2 0, E3 0, E4 0, E5 0, E6 0} C_DIS
   SPTP {A1 10.417, A2 -61.465, A3 83.836, A4 87.308, A5 -57.077, A6 0.000, E1 1201.82, E2 0, E3 0, E4 0, E5 0, E6 0} C_DIS
   SPTP {A1 10.268, A2 -61.945, A3 83.987, A4 88.436, A5 -56.152, A6 0.000, E1 1202, E2 0, E3 0, E4 0, E5 0, E6 0} C_DIS
   SPTP {A1 10.107, A2 -62.425, A3 84.142, A4 89.579, A5 -55.213, A6 0.000, E1 1202.15, E2 0, E3 0, E4 0, E5 0, E6 0} C_DIS
   SPTP {A1 9.934, A2 -62.905, A3 84.301, A4 90.740, A5 -54.264, A6 0.000, E1 1202.28, E2 0, E3 0, E4 0, E5 0, E6 0} C_DIS
   SPTP {A1 9.749, A2 -63.385, A3 84.464, A4 91.921, A5 -53.303, A6 0.000, E1 1202.36, E2 0, E3 0, E4 0, E5 0, E6 0} C_DIS
   SPTP {A1 9.553, A2 -63.865, A3 84.629, A4 93.124, A5 -52.330, A6 0.000, E1 1202.42, E2 0, E3 0, E4 0, E5 0, E6 0} C_DIS
   SPTP {A1 9.344, A2 -64.344, A3 84.798, A4 94.352, A5 -51.347, A6 0.000, E1 1202.44, E2 0, E3 0, E4 0, E5 0, E6 0} C_DIS
   SPTP {A1 9.123, A2 -64.820, A3 84.969, A4 95.607, A5 -50.354, A6 0.000, E1 1202.41, E2 0, E3 0, E4 0, E5 0, E6 0} C_DIS
   SPTP {A1 8.890, A2 -65.294, A3 85.141, A4 96.893, A5 -49.353, A6 0.000, E1 1202.35, E2 0, E3 0, E4 0, E5 0, E6 0} C_DIS
   SPTP {A1 8.645, A2 -65.765, A3 85.314, A4 98.212, A5 -48.346, A6 0.000, E1 1202.24, E2 0, E3 0, E4 0, E5 0, E6 0} C_DIS
   SPTP {A1 8.387, A2 -66.232, A3 85.488, A4 99.569, A5 -47.333, A6 0.000, E1 1202.08, E2 0, E3 0, E4 0, E5 0, E6 0} C_DIS
   SPTP {A1 8.118, A2 -66.695, A3 85.662, A4 100.967, A5 -46.317, A6 0.000, E1 1201.87, E2 0, E3 0, E4 0, E5 0, E6 0} C_DIS
   SPTP {A1 7.837, A2 -67.151, A3 85.833, A4 102.410, A5 -45.301, A6 0.000, E1 1201.6, E2 0, E3 0, E4 0, E5 0, E6 0} C_DIS
   SPTP {A1 7.533, A2 -67.610, A3 85.925, A4 104.243, A5 -44.229, A6 0.000, E1 1201.1, E2 0, E3 0, E4 0, E5 0, E6 0} C_DIS
   SPTP {A1 7.211, A2 -68.061, A3 85.982, A4 106.287, A5 -43.151, A6 0.000, E1 1200.44, E2 0, E3 0, E4 0, E5 0, E6 0} C_DIS
   SPTP {A1 6.874, A2 -68.501, A3 86.035, A4 108.410, A5 -42.093, A6 0.000, E1 1199.7, E2 0, E3 0, E4 0, E5 0, E6 0} C_DIS
   SPTP {A1 6.522, A2 -68.930, A3 86.085, A4 110.619, A5 -41.056, A6 0.000, E1 1198.86, E2 0, E3 0, E4 0, E5 0, E6 0} C_DIS
   SPTP {A1 6.156, A2 -69.347, A3 86.131, A4 112.917, A5 -40.049, A6 0.000, E1 1197.93, E2 0, E3 0, E4 0, E5 0, E6 0} C_DIS
   SPTP {A1 5.778, A2 -69.750, A3 86.173, A4 115.310, A5 -39.074, A6 0.000, E1 1196.89, E2 0, E3 0, E4 0, E5 0, E6 0} C_DIS
   SPTP {A1 5.388, A2 -70.139, A3 86.208, A4 117.799, A5 -38.141, A6 0.000, E1 1195.76, E2 0, E3 0, E4 0, E5 0, E6 0} C_DIS
   SPTP {A1 4.987, A2 -70.511, A3 86.237, A4 120.386, A5 -37.256, A6 0.000, E1 1194.53, E2 0, E3 0, E4 0, E5 0, E6 0} C_DIS
   SPTP {A1 4.577, A2 -70.868, A3 86.258, A4 123.068, A5 -36.426, A6 0.000, E1 1193.21, E2 0, E3 0, E4 0, E5 0, E6 0} C_DIS
   SPTP {A1 4.160, A2 -71.207, A3 86.273, A4 125.842, A5 -35.657, A6 0.000, E1 1191.79, E2 0, E3 0, E4 0, E5 0, E6 0} C_DIS
   SPTP {A1 3.737, A2 -71.529, A3 86.281, A4 128.701, A5 -34.954, A6 0.000, E1 1190.3, E2 0, E3 0, E4 0, E5 0, E6 0} C_DIS
   SPTP {A1 3.307, A2 -71.836, A3 86.285, A4 131.641, A5 -34.316, A6 0.000, E1 1188.73, E2 0, E3 0, E4 0, E5 0, E6 0} C_DIS
   SPTP {A1 2.874, A2 -72.125, A3 86.281, A4 134.645, A5 -33.756, A6 0.000, E1 1187.11, E2 0, E3 0, E4 0, E5 0, E6 0} C_DIS
   SPTP {A1 2.442, A2 -72.406, A3 86.306, A4 137.622, A5 -33.223, A6 0.000, E1 1185.55, E2 0, E3 0, E4 0, E5 0, E6 0} C_DIS
   SPTP {A1 2.006, A2 -72.783, A3 86.745, A4 139.794, A5 -32.083, A6 0.000, E1 1185, E2 0, E3 0, E4 0, E5 0, E6 0} C_DIS
   SPTP {A1 1.573, A2 -73.149, A3 87.192, A4 142.042, A5 -30.967, A6 0.000, E1 1184.38, E2 0, E3 0, E4 0, E5 0, E6 0} C_DIS
   SPTP {A1 1.143, A2 -73.503, A3 87.645, A4 144.367, A5 -29.876, A6 0.000, E1 1183.68, E2 0, E3 0, E4 0, E5 0, E6 0} C_DIS
   SPTP {A1 0.723, A2 -73.845, A3 88.105, A4 146.756, A5 -28.819, A6 0.000, E1 1182.94, E2 0, E3 0, E4 0, E5 0, E6 0} C_DIS
   SPTP {A1 0.315, A2 -74.175, A3 88.569, A4 149.192, A5 -27.800, A6 0.000, E1 1182.16, E2 0, E3 0, E4 0, E5 0, E6 0} C_DIS
   SPTP {A1 -0.077, A2 -74.494, A3 89.041, A4 151.656, A5 -26.821, A6 0.000, E1 1181.38, E2 0, E3 0, E4 0, E5 0, E6 0} C_DIS
   SPTP {A1 -0.447, A2 -74.802, A3 89.520, A4 154.123, A5 -25.882, A6 0.000, E1 1180.62, E2 0, E3 0, E4 0, E5 0, E6 0} C_DIS
   SPTP {A1 -0.782, A2 -75.235, A3 90.620, A4 155.189, A5 -23.813, A6 0.000, E1 1181.28, E2 0, E3 0, E4 0, E5 0, E6 0} C_DIS
   SPTP {A1 -1.085, A2 -75.658, A3 91.806, A4 155.914, A5 -21.556, A6 0.000, E1 1182.29, E2 0, E3 0, E4 0, E5 0, E6 0} C_DIS
   SPTP {A1 -1.357, A2 -76.046, A3 92.977, A4 156.470, A5 -19.300, A6 0.000, E1 1183.48, E2 0, E3 0, E4 0, E5 0, E6 0} C_DIS
   SPTP {A1 -1.585, A2 -76.398, A3 94.126, A4 156.678, A5 -17.063, A6 0.000, E1 1185.05, E2 0, E3 0, E4 0, E5 0, E6 0} C_DIS
   SPTP {A1 -1.765, A2 -76.714, A3 95.255, A4 156.360, A5 -14.845, A6 0.000, E1 1187.17, E2 0, E3 0, E4 0, E5 0, E6 0} C_DIS
   SPTP {A1 -1.895, A2 -77.027, A3 97.023, A4 151.296, A5 -11.150, A6 0.000, E1 1194, E2 0, E3 0, E4 0, E5 0, E6 0} C_DIS
   SPTP {A1 -1.973, A2 -77.226, A3 98.795, A4 138.768, A5 -7.492, A6 0.000, E1 1208.29, E2 0, E3 0, E4 0, E5 0, E6 0} C_DIS
   SPTP {A1 -2.003, A2 -77.296, A3 100.445, A4 107.317, A5 -4.909, A6 0.000, E1 1241.51, E2 0, E3 0, E4 0, E5 0, E6 0} C_DIS
   SPTP {A1 -1.977, A2 -77.233, A3 101.967, A4 59.416, A5 -5.371, A6 0.000, E1 1291.19, E2 0, E3 0, E4 0, E5 0, E6 0} C_DIS
   SPTP {A1 -1.901, A2 -76.935, A3 103.590, A4 31.124, A5 -9.193, A6 0.000, E1 1321.29, E2 0, E3 0, E4 0, E5 0, E6 0} C_DIS
   SPTP {A1 -1.793, A2 -76.234, A3 105.283, A4 19.345, A5 -15.225, A6 0.000, E1 1334.88, E2 0, E3 0, E4 0, E5 0, E6 0} C_DIS
   SPTP {A1 -1.646, A2 -75.232, A3 106.623, A4 14.849, A5 -21.535, A6 0.000, E1 1341.17, E2 0, E3 0, E4 0, E5 0, E6 0} C_DIS
   SPTP {A1 -1.473, A2 -73.944, A3 107.598, A4 12.742, A5 -27.882, A6 0.000, E1 1345.08, E2 0, E3 0, E4 0, E5 0, E6 0} C_DIS
   SPTP {A1 -1.281, A2 -71.727, A3 108.242, A4 10.956, A5 -36.306, A6 0.000, E1 1348.99, E2 0, E3 0, E4 0, E5 0, E6 0} C_DIS
   SPTP {A1 -1.085, A2 -69.093, A3 108.189, A4 10.096, A5 -44.503, A6 0.000, E1 1351.97, E2 0, E3 0, E4 0, E5 0, E6 0} C_DIS
   SPTP {A1 -0.891, A2 -66.115, A3 107.434, A4 9.715, A5 -52.366, A6 0.000, E1 1354.49, E2 0, E3 0, E4 0, E5 0, E6 0} C_DIS
   SPTP {A1 -0.712, A2 -62.874, A3 105.987, A4 9.586, A5 -59.813, A6 0.000, E1 1356.79, E2 0, E3 0, E4 0, E5 0, E6 0} C_DIS
   SPTP {A1 -0.321, A2 -60.181, A3 104.345, A4 10.283, A5 -65.367, A6 0.000, E1 1359.18, E2 0, E3 0, E4 0, E5 0, E6 0} C_DIS
   SPTP {A1 0.102, A2 -57.481, A3 102.329, A4 11.181, A5 -70.440, A6 0.000, E1 1361.53, E2 0, E3 0, E4 0, E5 0, E6 0} C_DIS
   SPTP {A1 0.540, A2 -54.744, A3 99.926, A4 12.227, A5 -75.141, A6 0.000, E1 1363.84, E2 0, E3 0, E4 0, E5 0, E6 0} C_DIS
   SPTP {A1 0.990, A2 -51.997, A3 97.153, A4 13.416, A5 -79.457, A6 0.000, E1 1366.12, E2 0, E3 0, E4 0, E5 0, E6 0} C_DIS
   SPTP {A1 1.445, A2 -49.254, A3 94.032, A4 14.723, A5 -83.386, A6 0.000, E1 1368.37, E2 0, E3 0, E4 0, E5 0, E6 0} C_DIS
   SPTP {A1 1.904, A2 -46.522, A3 90.572, A4 16.150, A5 -86.935, A6 0.000, E1 1370.6, E2 0, E3 0, E4 0, E5 0, E6 0} C_DIS
   SPTP {A1 2.369, A2 -43.796, A3 86.771, A4 17.713, A5 -90.112, A6 0.000, E1 1372.78, E2 0, E3 0, E4 0, E5 0, E6 0} C_DIS
   SPTP {A1 2.835, A2 -41.070, A3 82.627, A4 19.393, A5 -92.927, A6 0.000, E1 1374.89, E2 0, E3 0, E4 0, E5 0, E6 0} C_DIS
   SPTP {A1 3.298, A2 -38.323, A3 78.121, A4 21.180, A5 -95.388, A6 0.000, E1 1376.92, E2 0, E3 0, E4 0, E5 0, E6 0} C_DIS
   SPTP {A1 3.755, A2 -35.524, A3 73.210, A4 23.065, A5 -97.501, A6 0.000, E1 1378.82, E2 0, E3 0, E4 0, E5 0, E6 0} C_DIS
   SPTP {A1 4.297, A2 -34.795, A3 71.494, A4 25.177, A5 -97.877, A6 0.000, E1 1380.25, E2 0, E3 0, E4 0, E5 0, E6 0} C_DIS
   SPTP {A1 4.860, A2 -34.675, A3 70.726, A4 27.406, A5 -97.772, A6 0.000, E1 1381.42, E2 0, E3 0, E4 0, E5 0, E6 0} C_DIS
   SPTP {A1 5.413, A2 -34.533, A3 69.865, A4 29.690, A5 -97.637, A6 0.000, E1 1382.44, E2 0, E3 0, E4 0, E5 0, E6 0} C_DIS
   SPTP {A1 5.948, A2 -34.470, A3 69.098, A4 31.986, A5 -97.418, A6 0.000, E1 1383.28, E2 0, E3 0, E4 0, E5 0, E6 0} C_DIS
   SPTP {A1 6.427, A2 -35.130, A3 69.577, A4 34.110, A5 -96.740, A6 0.000, E1 1383.7, E2 0, E3 0, E4 0, E5 0, E6 0} C_DIS
   SPTP {A1 6.898, A2 -35.741, A3 69.930, A4 36.271, A5 -96.051, A6 0.000, E1 1383.99, E2 0, E3 0, E4 0, E5 0, E6 0} C_DIS
